# B&R Automation Studio project ConveyorTrackingSolution
Automation Studio 6.3.1.32; technology packages: mappMotion 6.4.1, OpcUaCs 6.3.1

## Configuration Config1

CPU 5APC3100.KBU3-000, AutomationRuntime 6.3.4, Build 11.3.0, Vc 

### Task classes (Cpu.sw)
```
Cyclic#1 (cycle 2000 us, tolerance 0 us):
  MovePrg <- MovePrg.prg
  ParChange <- ParChange.prg
DataObjects: McAcpSys
NcDataObjects: McDriveLog
Binaries: McAcpDrv, udbdef, McAcpSim, TCData, McProfGen, McMechSys, FWRules, ArSvcReg, BRRole, sysconf, iomap, TrkFrmSel, Config_3, Config_9, Config_4, Role, ashwac, Config_10, asfw, Config_5, Config_6, UaCsConfig, Config_8, Config_1, Hierarchy, ashwd, Config_11, Config_7, User, arconfig, Config_2, CommonFeat
Libraries: powerlnk, AsArProf, AsIecCon, fileio, AsIO, UaCoal, AsMem, astime, runtime, AsEPL, DataObj, brsystem, UaCoalPrv, SYS_LIB, MpBase, McBase, MpAxis, McAcpAx, McPathGen, McPureVAx, McAxGroup, McAxis, McProgInt, McTrkPath, MpRobotics
```

### Hardware
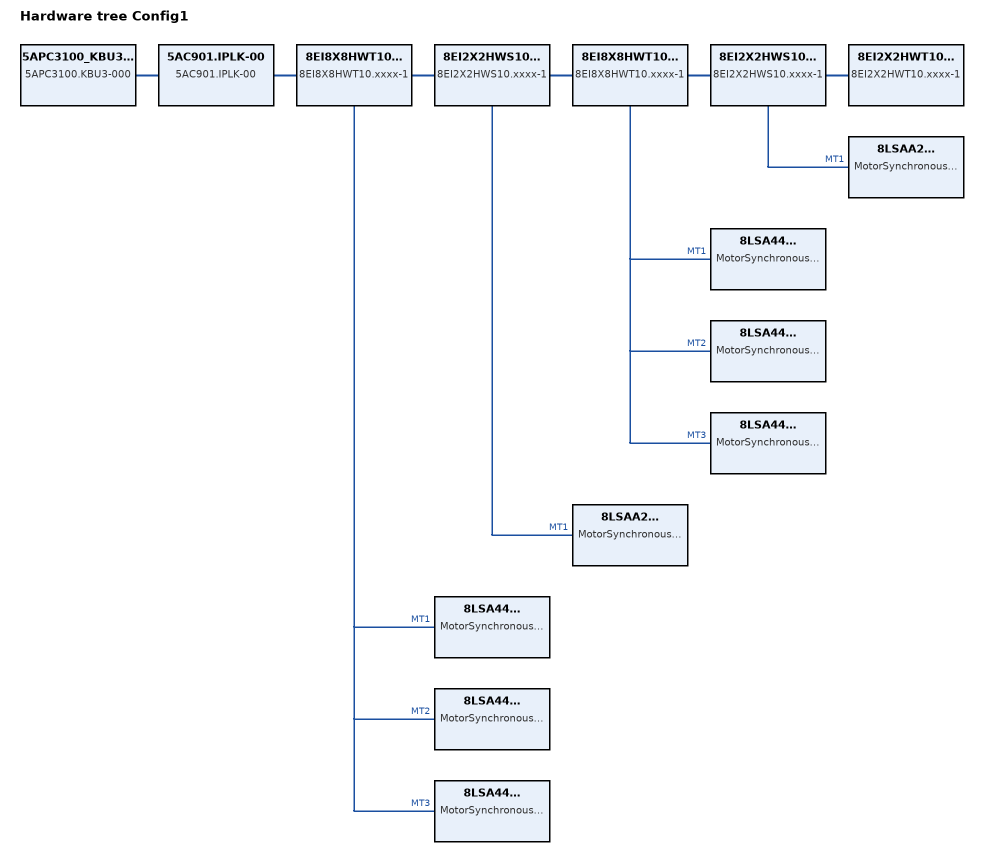
```
5AC901.IPLK-00 : 5AC901.IPLK-00 v2.1.0.0  [SL -> 5APC3100_KBU3_000.SL2]
5APC3100_KBU3_000 : 5APC3100.KBU3-000 v2.2.7.0
  Connector IF3:
    AssignedOperatingSystem = ARemb
    ActivateDevice = 1
  Connector IF4:
    AssignedOperatingSystem = ARemb
    ActivateDevice = 1
  Connector IF5:
    AssignedOperatingSystem = ARemb
  Connector IF6:
    AssignedOperatingSystem = ARemb
  Connector IF7:
    AssignedOperatingSystem = ARemb
  Connector IF8:
    AssignedOperatingSystem = ARemb
  ConfigurationID = ConveyorTrackingSolution_Config1
  Simulation = 1
  Cyclic1Duration = 2000
  Cyclic1Tolerance = 0
  FileDevice1
  FileDeviceName1 = USER
  FileDevicePath1 = USER_PATH
  FileDevice2
  FileDeviceName2 = CNC_PrgDir
  FileDevicePath2 = USER_PATH  // No simulation: use  USER_PATH   ;        Simulation: use    USER_PATH\..\..\..\..\..\Logical\CopyToUserPartition    to directly access the current progam state
8EI2X2HWS10.xxxx-1-QC_D4r1100R_1 : 8EI2X2HWS10.xxxx-1 v2.3.2.0 (NodeNumber=2)  [PLK1 -> 8EI8X8HWT10.xxxx-1-Q1-Q2-Q3_D4r1100R_1.PLK2 [Cable Type=PowerlinkCable, Length=10, Version=1.0.0.3]; PLK2 -> 8EI8X8HWT10.xxxx-1-Q1-Q2-Q3_D4r1100R_2.PLK1 [Cable Type=PowerlinkCable, Length=10, Version=1.0.0.3]]
  DriveConfiguration/Encoder/EncoderX41:
    InterfaceType = EnDat
  DriveConfiguration/Channel[1]/RealAxis:
    AxisReference = gAxisQC_D4r1100R_1
  DriveConfiguration/Channel[1]/RealAxis/MechanicalElements/Gearbox:
    InputIsReadOnly = 1
    Input = 10
    OutputIsReadOnly = 1
  DriveConfiguration/Channel[1]/RealAxis/MechanicalElements/RotaryToLinearTransformation:
    ReferenceDistanceIsReadOnly = 1
    ReferenceDistance = 360
  DriveConfiguration/Channel[1]/RealAxis/Controller:
    ModeIsReadOnly = 1
    Mode = PositionControllerWithTorqueFeedForward
  DriveConfiguration/Channel[1]/RealAxis/Controller/Mode/Position:
    ProportionalGainIsReadOnly = 1
    ProportionalGain = 80.0
    IntegrationTimeIsReadOnly = 1
  DriveConfiguration/Channel[1]/RealAxis/Controller/Mode/Speed:
    ProportionalGainIsReadOnly = 1
    IntegrationTimeIsReadOnly = 1
    FilterTimeIsReadOnly = 1
  DriveConfiguration/Channel[1]/RealAxis/Controller/Mode:
    FeedForwardIsReadOnly = 1
    FeedForward = CyclicValueFromAxesGroup
  DriveConfiguration/Channel[1]/RealAxis/Controller/Mode/LoopFilters:
    LoopFilterXIsReadOnly = 1
  DriveConfiguration/Channel[1]/RealAxis/Homing:
    Mode = Absolute
    RestorePositionVariable = 
  DriveConfiguration/Channel[1]/RealAxis/StopReaction:
    DriveError = CyclicDecelerationFromAxesGroup
  DriveConfiguration/Channel[1]/RealAxis/MovementErrorLimits:
    PositionError = 0.5
  DriveConfiguration/Channel[1]/RealAxis:
    JerkFilterIsReadOnly = 1
    JerkFilter = Used
  DriveConfiguration/Channel[1]/RealAxis/JerkFilter:
    JerkTimeMin = 0.06
    JerkTime = 0.06
8EI2X2HWS10.xxxx-1-QC_D4r1100R_2 : 8EI2X2HWS10.xxxx-1 v2.3.2.0 (NodeNumber=4)  [PLK1 -> 8EI8X8HWT10.xxxx-1-Q1-Q2-Q3_D4r1100R_2.PLK2 [Cable Type=PowerlinkCable, Length=10, Version=1.0.0.3]; PLK2 -> 8EI2X2HWT10.xxxx-1.PLK1 [Cable Type=PowerlinkCable, Length=10, Version=1.0.0.3]]
  DriveConfiguration/Encoder/EncoderX41:
    InterfaceType = EnDat
  DriveConfiguration/Channel[1]/RealAxis:
    AxisReference = gAxisQC_D4r1100R_2
  DriveConfiguration/Channel[1]/RealAxis/MechanicalElements/Gearbox:
    InputIsReadOnly = 1
    Input = 10
    OutputIsReadOnly = 1
  DriveConfiguration/Channel[1]/RealAxis/MechanicalElements/RotaryToLinearTransformation:
    ReferenceDistanceIsReadOnly = 1
    ReferenceDistance = 360
  DriveConfiguration/Channel[1]/RealAxis/Controller:
    ModeIsReadOnly = 1
    Mode = PositionControllerWithTorqueFeedForward
  DriveConfiguration/Channel[1]/RealAxis/Controller/Mode/Position:
    ProportionalGainIsReadOnly = 1
    ProportionalGain = 80.0
    IntegrationTimeIsReadOnly = 1
  DriveConfiguration/Channel[1]/RealAxis/Controller/Mode/Speed:
    ProportionalGainIsReadOnly = 1
    IntegrationTimeIsReadOnly = 1
    FilterTimeIsReadOnly = 1
  DriveConfiguration/Channel[1]/RealAxis/Controller/Mode:
    FeedForwardIsReadOnly = 1
    FeedForward = CyclicValueFromAxesGroup
  DriveConfiguration/Channel[1]/RealAxis/Controller/Mode/LoopFilters:
    LoopFilterXIsReadOnly = 1
  DriveConfiguration/Channel[1]/RealAxis/Homing:
    Mode = Absolute
    RestorePositionVariable = 
  DriveConfiguration/Channel[1]/RealAxis/StopReaction:
    DriveError = CyclicDecelerationFromAxesGroup
  DriveConfiguration/Channel[1]/RealAxis/MovementErrorLimits:
    PositionError = 0.5
  DriveConfiguration/Channel[1]/RealAxis:
    JerkFilterIsReadOnly = 1
    JerkFilter = Used
  DriveConfiguration/Channel[1]/RealAxis/JerkFilter:
    JerkTimeMin = 0.06
    JerkTime = 0.06
8EI2X2HWT10.xxxx-1 : 8EI2X2HWT10.xxxx-1 v2.4.0.0 (NodeNumber=5)  [PLK1 -> 8EI2X2HWS10.xxxx-1-QC_D4r1100R_2.PLK2 [Cable Type=PowerlinkCable, Length=10, Version=1.0.0.3]]
  DriveConfiguration/Channel[1]/RealAxis:
    AxisReference = gAxis_Conveyor_1
  DriveConfiguration/Channel[2]/RealAxis:
    AxisReference = gAxis_Conveyor_2
8EI8X8HWT10.xxxx-1-Q1-Q2-Q3_D4r1100R_1 : 8EI8X8HWT10.xxxx-1 v2.3.2.0 (NodeNumber=1)  [PLK1 -> 5AC901.IPLK-00.IF1 [Cable Type=PowerlinkCable, Length=10, Version=1.0.0.3]; PLK2 -> 8EI2X2HWS10.xxxx-1-QC_D4r1100R_1.PLK1 [Cable Type=PowerlinkCable, Length=10, Version=1.0.0.3]; MT2 -> 8LSA44.DB060S200-3_Q2_D4r1100R_1.MT; MT3 -> 8LSA44.DB060S200-3_Q3_D4r1100R_1.MT]
  DriveConfiguration/Encoder/EncoderX41:
    InterfaceType = EnDat
  DriveConfiguration/Encoder/EncoderX42:
    InterfaceType = EnDat
  DriveConfiguration/Encoder/EncoderX43:
    InterfaceType = EnDat
  DriveConfiguration/Channel[1]/RealAxis:
    AxisReference = gAxisQ1_D4r1100R_1
  DriveConfiguration/Channel[1]/RealAxis/MechanicalElements/Gearbox:
    InputIsReadOnly = 1
    Input = 28
    OutputIsReadOnly = 1
  DriveConfiguration/Channel[1]/RealAxis/MechanicalElements/RotaryToLinearTransformation:
    ReferenceDistanceIsReadOnly = 1
    ReferenceDistance = 360
  DriveConfiguration/Channel[1]/RealAxis/Controller:
    ModeIsReadOnly = 1
    Mode = PositionControllerWithTorqueFeedForward
  DriveConfiguration/Channel[1]/RealAxis/Controller/Mode/Position:
    ProportionalGainIsReadOnly = 1
    ProportionalGain = 150.0
    IntegrationTimeIsReadOnly = 1
  DriveConfiguration/Channel[1]/RealAxis/Controller/Mode/Speed:
    ProportionalGainIsReadOnly = 1
    ProportionalGain = 7.5
    IntegrationTimeIsReadOnly = 1
    FilterTimeIsReadOnly = 1
  DriveConfiguration/Channel[1]/RealAxis/Controller/Mode:
    FeedForwardIsReadOnly = 1
    FeedForward = CyclicValueFromAxesGroup
  DriveConfiguration/Channel[1]/RealAxis/Controller/Mode/LoopFilters:
    LoopFilterXIsReadOnly = 1
  DriveConfiguration/Channel[1]/RealAxis/Homing:
    Mode = Absolute
    RestorePositionVariable = 
  DriveConfiguration/Channel[1]/RealAxis/StopReaction:
    DriveError = CyclicDecelerationFromAxesGroup
  DriveConfiguration/Channel[1]/RealAxis/MovementErrorLimits:
    PositionError = 0.5
  DriveConfiguration/Channel[1]/RealAxis:
    JerkFilterIsReadOnly = 1
    JerkFilter = Used
  DriveConfiguration/Channel[1]/RealAxis/JerkFilter:
    JerkTimeMin = 0.06
    JerkTime = 0.06
  DriveConfiguration/Channel[2]/RealAxis:
    AxisReference = gAxisQ2_D4r1100R_1
  DriveConfiguration/Channel[2]/RealAxis/MechanicalElements/Gearbox:
    InputIsReadOnly = 1
    Input = 28
    OutputIsReadOnly = 1
  DriveConfiguration/Channel[2]/RealAxis/MechanicalElements/RotaryToLinearTransformation:
    ReferenceDistanceIsReadOnly = 1
    ReferenceDistance = 360
  DriveConfiguration/Channel[2]/RealAxis/Controller:
    ModeIsReadOnly = 1
    Mode = PositionControllerWithTorqueFeedForward
  DriveConfiguration/Channel[2]/RealAxis/Controller/Mode/Position:
    ProportionalGainIsReadOnly = 1
    ProportionalGain = 150.0
    IntegrationTimeIsReadOnly = 1
  DriveConfiguration/Channel[2]/RealAxis/Controller/Mode/Speed:
    ProportionalGainIsReadOnly = 1
    ProportionalGain = 7.5
    IntegrationTimeIsReadOnly = 1
    FilterTimeIsReadOnly = 1
  DriveConfiguration/Channel[2]/RealAxis/Controller/Mode:
    FeedForwardIsReadOnly = 1
    FeedForward = CyclicValueFromAxesGroup
  DriveConfiguration/Channel[2]/RealAxis/Controller/Mode/LoopFilters:
    LoopFilterXIsReadOnly = 1
  DriveConfiguration/Channel[2]/RealAxis/Homing:
    Mode = Absolute
    RestorePositionVariable = 
  DriveConfiguration/Channel[2]/RealAxis/StopReaction:
    DriveError = CyclicDecelerationFromAxesGroup
  DriveConfiguration/Channel[2]/RealAxis/MovementErrorLimits:
    PositionError = 0.5
  DriveConfiguration/Channel[2]/RealAxis:
    JerkFilterIsReadOnly = 1
    JerkFilter = Used
  DriveConfiguration/Channel[2]/RealAxis/JerkFilter:
    JerkTimeMin = 0.06
    JerkTime = 0.06
  DriveConfiguration/Channel[3]/RealAxis:
    AxisReference = gAxisQ3_D4r1100R_1
  DriveConfiguration/Channel[3]/RealAxis/MechanicalElements/Gearbox:
    InputIsReadOnly = 1
    Input = 28
    OutputIsReadOnly = 1
  DriveConfiguration/Channel[3]/RealAxis/MechanicalElements/RotaryToLinearTransformation:
    ReferenceDistanceIsReadOnly = 1
    ReferenceDistance = 360
  DriveConfiguration/Channel[3]/RealAxis/Controller:
    ModeIsReadOnly = 1
    Mode = PositionControllerWithTorqueFeedForward
  DriveConfiguration/Channel[3]/RealAxis/Controller/Mode/Position:
    ProportionalGainIsReadOnly = 1
    ProportionalGain = 150.0
    IntegrationTimeIsReadOnly = 1
  DriveConfiguration/Channel[3]/RealAxis/Controller/Mode/Speed:
    ProportionalGainIsReadOnly = 1
    ProportionalGain = 7.5
    IntegrationTimeIsReadOnly = 1
    FilterTimeIsReadOnly = 1
  DriveConfiguration/Channel[3]/RealAxis/Controller/Mode:
    FeedForwardIsReadOnly = 1
    FeedForward = CyclicValueFromAxesGroup
  DriveConfiguration/Channel[3]/RealAxis/Controller/Mode/LoopFilters:
    LoopFilterXIsReadOnly = 1
  DriveConfiguration/Channel[3]/RealAxis/Homing:
    Mode = Absolute
    RestorePositionVariable = 
  DriveConfiguration/Channel[3]/RealAxis/StopReaction:
    DriveError = CyclicDecelerationFromAxesGroup
  DriveConfiguration/Channel[3]/RealAxis/MovementErrorLimits:
    PositionError = 0.5
  DriveConfiguration/Channel[3]/RealAxis:
    JerkFilterIsReadOnly = 1
    JerkFilter = Used
  DriveConfiguration/Channel[3]/RealAxis/JerkFilter:
    JerkTimeMin = 0.06
    JerkTime = 0.06
8EI8X8HWT10.xxxx-1-Q1-Q2-Q3_D4r1100R_2 : 8EI8X8HWT10.xxxx-1 v2.3.2.0 (NodeNumber=3)  [PLK1 -> 8EI2X2HWS10.xxxx-1-QC_D4r1100R_1.PLK2 [Cable Type=PowerlinkCable, Length=10, Version=1.0.0.3]; PLK2 -> 8EI2X2HWS10.xxxx-1-QC_D4r1100R_2.PLK1 [Cable Type=PowerlinkCable, Length=10, Version=1.0.0.3]; MT2 -> 8LSA44.DB060S200-3_Q2_D4r1100R_2.MT; MT3 -> 8LSA44.DB060S200-3_Q3_D4r1100R_2.MT]
  DriveConfiguration/Encoder/EncoderX41:
    InterfaceType = EnDat
  DriveConfiguration/Encoder/EncoderX42:
    InterfaceType = EnDat
  DriveConfiguration/Encoder/EncoderX43:
    InterfaceType = EnDat
  DriveConfiguration/Channel[1]/RealAxis:
    AxisReference = gAxisQ1_D4r1100R_2
  DriveConfiguration/Channel[1]/RealAxis/MechanicalElements/Gearbox:
    InputIsReadOnly = 1
    Input = 28
    OutputIsReadOnly = 1
  DriveConfiguration/Channel[1]/RealAxis/MechanicalElements/RotaryToLinearTransformation:
    ReferenceDistanceIsReadOnly = 1
    ReferenceDistance = 360
  DriveConfiguration/Channel[1]/RealAxis/Controller:
    ModeIsReadOnly = 1
    Mode = PositionControllerWithTorqueFeedForward
  DriveConfiguration/Channel[1]/RealAxis/Controller/Mode/Position:
    ProportionalGainIsReadOnly = 1
    ProportionalGain = 150.0
    IntegrationTimeIsReadOnly = 1
  DriveConfiguration/Channel[1]/RealAxis/Controller/Mode/Speed:
    ProportionalGainIsReadOnly = 1
    ProportionalGain = 7.5
    IntegrationTimeIsReadOnly = 1
    FilterTimeIsReadOnly = 1
  DriveConfiguration/Channel[1]/RealAxis/Controller/Mode:
    FeedForwardIsReadOnly = 1
    FeedForward = CyclicValueFromAxesGroup
  DriveConfiguration/Channel[1]/RealAxis/Controller/Mode/LoopFilters:
    LoopFilterXIsReadOnly = 1
  DriveConfiguration/Channel[1]/RealAxis/Homing:
    Mode = Absolute
    RestorePositionVariable = 
  DriveConfiguration/Channel[1]/RealAxis/StopReaction:
    DriveError = CyclicDecelerationFromAxesGroup
  DriveConfiguration/Channel[1]/RealAxis/MovementErrorLimits:
    PositionError = 0.5
  DriveConfiguration/Channel[1]/RealAxis:
    JerkFilterIsReadOnly = 1
    JerkFilter = Used
  DriveConfiguration/Channel[1]/RealAxis/JerkFilter:
    JerkTimeMin = 0.06
    JerkTime = 0.06
  DriveConfiguration/Channel[2]/RealAxis:
    AxisReference = gAxisQ2_D4r1100R_2
  DriveConfiguration/Channel[2]/RealAxis/MechanicalElements/Gearbox:
    InputIsReadOnly = 1
    Input = 28
    OutputIsReadOnly = 1
  DriveConfiguration/Channel[2]/RealAxis/MechanicalElements/RotaryToLinearTransformation:
    ReferenceDistanceIsReadOnly = 1
    ReferenceDistance = 360
  DriveConfiguration/Channel[2]/RealAxis/Controller:
    ModeIsReadOnly = 1
    Mode = PositionControllerWithTorqueFeedForward
  DriveConfiguration/Channel[2]/RealAxis/Controller/Mode/Position:
    ProportionalGainIsReadOnly = 1
    ProportionalGain = 150.0
    IntegrationTimeIsReadOnly = 1
  DriveConfiguration/Channel[2]/RealAxis/Controller/Mode/Speed:
    ProportionalGainIsReadOnly = 1
    ProportionalGain = 7.5
    IntegrationTimeIsReadOnly = 1
    FilterTimeIsReadOnly = 1
  DriveConfiguration/Channel[2]/RealAxis/Controller/Mode:
    FeedForwardIsReadOnly = 1
    FeedForward = CyclicValueFromAxesGroup
  DriveConfiguration/Channel[2]/RealAxis/Controller/Mode/LoopFilters:
    LoopFilterXIsReadOnly = 1
  DriveConfiguration/Channel[2]/RealAxis/Homing:
    Mode = Absolute
    RestorePositionVariable = 
  DriveConfiguration/Channel[2]/RealAxis/StopReaction:
    DriveError = CyclicDecelerationFromAxesGroup
  DriveConfiguration/Channel[2]/RealAxis/MovementErrorLimits:
    PositionError = 0.5
  DriveConfiguration/Channel[2]/RealAxis:
    JerkFilterIsReadOnly = 1
    JerkFilter = Used
  DriveConfiguration/Channel[2]/RealAxis/JerkFilter:
    JerkTimeMin = 0.06
    JerkTime = 0.06
  DriveConfiguration/Channel[3]/RealAxis:
    AxisReference = gAxisQ3_D4r1100R_2
  DriveConfiguration/Channel[3]/RealAxis/MechanicalElements/Gearbox:
    InputIsReadOnly = 1
    Input = 28
    OutputIsReadOnly = 1
  DriveConfiguration/Channel[3]/RealAxis/MechanicalElements/RotaryToLinearTransformation:
    ReferenceDistanceIsReadOnly = 1
    ReferenceDistance = 360
  DriveConfiguration/Channel[3]/RealAxis/Controller:
    ModeIsReadOnly = 1
    Mode = PositionControllerWithTorqueFeedForward
  DriveConfiguration/Channel[3]/RealAxis/Controller/Mode/Position:
    ProportionalGainIsReadOnly = 1
    ProportionalGain = 150.0
    IntegrationTimeIsReadOnly = 1
  DriveConfiguration/Channel[3]/RealAxis/Controller/Mode/Speed:
    ProportionalGainIsReadOnly = 1
    ProportionalGain = 7.5
    IntegrationTimeIsReadOnly = 1
    FilterTimeIsReadOnly = 1
  DriveConfiguration/Channel[3]/RealAxis/Controller/Mode:
    FeedForwardIsReadOnly = 1
    FeedForward = CyclicValueFromAxesGroup
  DriveConfiguration/Channel[3]/RealAxis/Controller/Mode/LoopFilters:
    LoopFilterXIsReadOnly = 1
  DriveConfiguration/Channel[3]/RealAxis/Homing:
    Mode = Absolute
    RestorePositionVariable = 
  DriveConfiguration/Channel[3]/RealAxis/StopReaction:
    DriveError = CyclicDecelerationFromAxesGroup
  DriveConfiguration/Channel[3]/RealAxis/MovementErrorLimits:
    PositionError = 0.5
  DriveConfiguration/Channel[3]/RealAxis:
    JerkFilterIsReadOnly = 1
    JerkFilter = Used
  DriveConfiguration/Channel[3]/RealAxis/JerkFilter:
    JerkTimeMin = 0.06
    JerkTime = 0.06
8LSA44.DB060S200-3_Q1_D4r1100R_1 : MotorSynchronous_any v2.2.1.0  [MT -> 8EI8X8HWT10.xxxx-1-Q1-Q2-Q3_D4r1100R_1.MT1]
  M1/MotorParameters:
    MOTOR_POLEPAIRS = 5
    MOTOR_SPEED_RATED = 6000
    MOTOR_SPEED_MAX = 12000
    MOTOR_VOLTAGE_RATED = 400
    MOTOR_CURR_RATED = 3.7
    MOTOR_CURR_STALL = 7.4
    MOTOR_CURR_MAX = 43.8
    MOTOR_TORQ_RATED = 3
    MOTOR_TORQ_STALL = 6
    MOTOR_TORQ_MAX = 22.8
    MOTOR_VOLTAGE_CONST = 49.22
    MOTOR_TORQ_CONST = 0.81
    MOTOR_STATOR_RESISTANCE = 0.863
    MOTOR_STATOR_INDUCTANCE = 6.2
    MOTOR_INERTIA = 2.73
    VoltageLimitation = Used
  M1/MotorParameters/VoltageLimitation:
    MOTOR_UDC_MAX = 1000
  M1/MotorParameters/EncoderMounting:
    Angle = StoredOnEncoder
  M1/MotorParameters/TemperatureSensor:
    MOTOR_TEMPSENS_LIM = 130
    TemperatureSensorInterface = EncoderConnectorDigital
    MOTOR_TEMPSENS_PAR1 = 30
    MOTOR_TEMPSENS_PAR2 = 254
    MOTOR_TEMPSENS_PAR3 = -29.72
    MOTOR_TEMPSENS_PAR4 = -4.58
    MOTOR_TEMPSENS_PAR5 = 20.33
    MOTOR_TEMPSENS_PAR6 = 45.18
    MOTOR_TEMPSENS_PAR7 = 69.96
    MOTOR_TEMPSENS_PAR8 = 94.71
    MOTOR_TEMPSENS_PAR9 = 119.6
    MOTOR_TEMPSENS_PAR10 = 149.11
  M1/MotorParameters/TemperatureModel:
    MOTOR_WIND_TEMP_MAX = 110
  M1/MotorParameters/TemperatureModel/Calculation:
    MOTOR_WIND_CROSS_SECT = 0.985
    MOTOR_TAU_THERM = 1800
  M1:
    Brake = Used
  M1/Brake:
    MOTOR_BRAKE_CURR_RATED = 0.83
    MOTOR_BRAKE_TORQ_RATED = 8
    MOTOR_BRAKE_ON_TIME = 0.038
    MOTOR_BRAKE_OFF_TIME = 0.055
    MOTOR_BRAKE_INERTIA = 0.69
  M1/Encoder:
    MOTOR_ENCOD_ATTR = 1
    MOTOR_ENCOD_INERTIA = 0.022
    TemperatureSensor = Used
  M1/Encoder/TemperatureSensor:
    MOTOR_ENCOD_TEMP_LIM = 129
  M1:
    Gearbox = UsedWithDynamicTorqueLimitation
  M1/Gearbox/GearRatio:
    Input = 28
  M1/Gearbox:
    MOTORGEAR_SPEED_MAX = 7500
    MOTORGEAR_TORQ_NOM = 126
    MOTORGEAR_TORQ_MAX = 126
    MOTORGEAR_INERTIA = 0.51
    MOTORGEAR_VISC_FRIC = 0.002
    MOTORGEAR_STAT_FRIC = 0.22
8LSA44.DB060S200-3_Q1_D4r1100R_2 : MotorSynchronous_any v2.2.1.0  [MT -> 8EI8X8HWT10.xxxx-1-Q1-Q2-Q3_D4r1100R_2.MT1]
  M1/MotorParameters:
    MOTOR_POLEPAIRS = 5
    MOTOR_SPEED_RATED = 6000
    MOTOR_SPEED_MAX = 12000
    MOTOR_VOLTAGE_RATED = 400
    MOTOR_CURR_RATED = 3.7
    MOTOR_CURR_STALL = 7.4
    MOTOR_CURR_MAX = 43.8
    MOTOR_TORQ_RATED = 3
    MOTOR_TORQ_STALL = 6
    MOTOR_TORQ_MAX = 22.8
    MOTOR_VOLTAGE_CONST = 49.22
    MOTOR_TORQ_CONST = 0.81
    MOTOR_STATOR_RESISTANCE = 0.863
    MOTOR_STATOR_INDUCTANCE = 6.2
    MOTOR_INERTIA = 2.73
    VoltageLimitation = Used
  M1/MotorParameters/VoltageLimitation:
    MOTOR_UDC_MAX = 1000
  M1/MotorParameters/EncoderMounting:
    Angle = StoredOnEncoder
  M1/MotorParameters/TemperatureSensor:
    MOTOR_TEMPSENS_LIM = 130
    TemperatureSensorInterface = EncoderConnectorDigital
    MOTOR_TEMPSENS_PAR1 = 30
    MOTOR_TEMPSENS_PAR2 = 254
    MOTOR_TEMPSENS_PAR3 = -29.72
    MOTOR_TEMPSENS_PAR4 = -4.58
    MOTOR_TEMPSENS_PAR5 = 20.33
    MOTOR_TEMPSENS_PAR6 = 45.18
    MOTOR_TEMPSENS_PAR7 = 69.96
    MOTOR_TEMPSENS_PAR8 = 94.71
    MOTOR_TEMPSENS_PAR9 = 119.6
    MOTOR_TEMPSENS_PAR10 = 149.11
  M1/MotorParameters/TemperatureModel:
    MOTOR_WIND_TEMP_MAX = 110
  M1/MotorParameters/TemperatureModel/Calculation:
    MOTOR_WIND_CROSS_SECT = 0.985
    MOTOR_TAU_THERM = 1800
  M1:
    Brake = Used
  M1/Brake:
    MOTOR_BRAKE_CURR_RATED = 0.83
    MOTOR_BRAKE_TORQ_RATED = 8
    MOTOR_BRAKE_ON_TIME = 0.038
    MOTOR_BRAKE_OFF_TIME = 0.055
    MOTOR_BRAKE_INERTIA = 0.69
  M1/Encoder:
    MOTOR_ENCOD_ATTR = 1
    MOTOR_ENCOD_INERTIA = 0.022
    TemperatureSensor = Used
  M1/Encoder/TemperatureSensor:
    MOTOR_ENCOD_TEMP_LIM = 129
  M1:
    Gearbox = UsedWithDynamicTorqueLimitation
  M1/Gearbox/GearRatio:
    Input = 28
  M1/Gearbox:
    MOTORGEAR_SPEED_MAX = 7500
    MOTORGEAR_TORQ_NOM = 126
    MOTORGEAR_TORQ_MAX = 126
    MOTORGEAR_INERTIA = 0.51
    MOTORGEAR_VISC_FRIC = 0.002
    MOTORGEAR_STAT_FRIC = 0.22
8LSA44.DB060S200-3_Q2_D4r1100R_1 : MotorSynchronous_any v2.2.1.0  [MT -> 8EI8X8HWT10.xxxx-1-Q1-Q2-Q3_D4r1100R_1.MT2]
  M1/MotorParameters:
    MOTOR_POLEPAIRS = 5
    MOTOR_SPEED_RATED = 6000
    MOTOR_SPEED_MAX = 12000
    MOTOR_VOLTAGE_RATED = 400
    MOTOR_CURR_RATED = 3.7
    MOTOR_CURR_STALL = 7.4
    MOTOR_CURR_MAX = 43.8
    MOTOR_TORQ_RATED = 3
    MOTOR_TORQ_STALL = 6
    MOTOR_TORQ_MAX = 22.8
    MOTOR_VOLTAGE_CONST = 49.22
    MOTOR_TORQ_CONST = 0.81
    MOTOR_STATOR_RESISTANCE = 0.863
    MOTOR_STATOR_INDUCTANCE = 6.2
    MOTOR_INERTIA = 2.73
    VoltageLimitation = Used
  M1/MotorParameters/VoltageLimitation:
    MOTOR_UDC_MAX = 1000
  M1/MotorParameters/EncoderMounting:
    Angle = StoredOnEncoder
  M1/MotorParameters/TemperatureSensor:
    MOTOR_TEMPSENS_LIM = 130
    TemperatureSensorInterface = EncoderConnectorDigital
    MOTOR_TEMPSENS_PAR1 = 30
    MOTOR_TEMPSENS_PAR2 = 254
    MOTOR_TEMPSENS_PAR3 = -29.72
    MOTOR_TEMPSENS_PAR4 = -4.58
    MOTOR_TEMPSENS_PAR5 = 20.33
    MOTOR_TEMPSENS_PAR6 = 45.18
    MOTOR_TEMPSENS_PAR7 = 69.96
    MOTOR_TEMPSENS_PAR8 = 94.71
    MOTOR_TEMPSENS_PAR9 = 119.6
    MOTOR_TEMPSENS_PAR10 = 149.11
  M1/MotorParameters/TemperatureModel:
    MOTOR_WIND_TEMP_MAX = 110
  M1/MotorParameters/TemperatureModel/Calculation:
    MOTOR_WIND_CROSS_SECT = 0.985
    MOTOR_TAU_THERM = 1800
  M1:
    Brake = Used
  M1/Brake:
    MOTOR_BRAKE_CURR_RATED = 0.83
    MOTOR_BRAKE_TORQ_RATED = 8
    MOTOR_BRAKE_ON_TIME = 0.038
    MOTOR_BRAKE_OFF_TIME = 0.055
    MOTOR_BRAKE_INERTIA = 0.69
  M1/Encoder:
    MOTOR_ENCOD_ATTR = 1
    MOTOR_ENCOD_INERTIA = 0.022
    TemperatureSensor = Used
  M1/Encoder/TemperatureSensor:
    MOTOR_ENCOD_TEMP_LIM = 129
  M1:
    Gearbox = UsedWithDynamicTorqueLimitation
  M1/Gearbox/GearRatio:
    Input = 28
  M1/Gearbox:
    MOTORGEAR_SPEED_MAX = 7500
    MOTORGEAR_TORQ_NOM = 126
    MOTORGEAR_TORQ_MAX = 126
    MOTORGEAR_INERTIA = 0.51
    MOTORGEAR_VISC_FRIC = 0.002
    MOTORGEAR_STAT_FRIC = 0.22
8LSA44.DB060S200-3_Q2_D4r1100R_2 : MotorSynchronous_any v2.2.1.0  [MT -> 8EI8X8HWT10.xxxx-1-Q1-Q2-Q3_D4r1100R_2.MT2]
  M1/MotorParameters:
    MOTOR_POLEPAIRS = 5
    MOTOR_SPEED_RATED = 6000
    MOTOR_SPEED_MAX = 12000
    MOTOR_VOLTAGE_RATED = 400
    MOTOR_CURR_RATED = 3.7
    MOTOR_CURR_STALL = 7.4
    MOTOR_CURR_MAX = 43.8
    MOTOR_TORQ_RATED = 3
    MOTOR_TORQ_STALL = 6
    MOTOR_TORQ_MAX = 22.8
    MOTOR_VOLTAGE_CONST = 49.22
    MOTOR_TORQ_CONST = 0.81
    MOTOR_STATOR_RESISTANCE = 0.863
    MOTOR_STATOR_INDUCTANCE = 6.2
    MOTOR_INERTIA = 2.73
    VoltageLimitation = Used
  M1/MotorParameters/VoltageLimitation:
    MOTOR_UDC_MAX = 1000
  M1/MotorParameters/EncoderMounting:
    Angle = StoredOnEncoder
  M1/MotorParameters/TemperatureSensor:
    MOTOR_TEMPSENS_LIM = 130
    TemperatureSensorInterface = EncoderConnectorDigital
    MOTOR_TEMPSENS_PAR1 = 30
    MOTOR_TEMPSENS_PAR2 = 254
    MOTOR_TEMPSENS_PAR3 = -29.72
    MOTOR_TEMPSENS_PAR4 = -4.58
    MOTOR_TEMPSENS_PAR5 = 20.33
    MOTOR_TEMPSENS_PAR6 = 45.18
    MOTOR_TEMPSENS_PAR7 = 69.96
    MOTOR_TEMPSENS_PAR8 = 94.71
    MOTOR_TEMPSENS_PAR9 = 119.6
    MOTOR_TEMPSENS_PAR10 = 149.11
  M1/MotorParameters/TemperatureModel:
    MOTOR_WIND_TEMP_MAX = 110
  M1/MotorParameters/TemperatureModel/Calculation:
    MOTOR_WIND_CROSS_SECT = 0.985
    MOTOR_TAU_THERM = 1800
  M1:
    Brake = Used
  M1/Brake:
    MOTOR_BRAKE_CURR_RATED = 0.83
    MOTOR_BRAKE_TORQ_RATED = 8
    MOTOR_BRAKE_ON_TIME = 0.038
    MOTOR_BRAKE_OFF_TIME = 0.055
    MOTOR_BRAKE_INERTIA = 0.69
  M1/Encoder:
    MOTOR_ENCOD_ATTR = 1
    MOTOR_ENCOD_INERTIA = 0.022
    TemperatureSensor = Used
  M1/Encoder/TemperatureSensor:
    MOTOR_ENCOD_TEMP_LIM = 129
  M1:
    Gearbox = UsedWithDynamicTorqueLimitation
  M1/Gearbox/GearRatio:
    Input = 28
  M1/Gearbox:
    MOTORGEAR_SPEED_MAX = 7500
    MOTORGEAR_TORQ_NOM = 126
    MOTORGEAR_TORQ_MAX = 126
    MOTORGEAR_INERTIA = 0.51
    MOTORGEAR_VISC_FRIC = 0.002
    MOTORGEAR_STAT_FRIC = 0.22
8LSA44.DB060S200-3_Q3_D4r1100R_1 : MotorSynchronous_any v2.2.1.0  [MT -> 8EI8X8HWT10.xxxx-1-Q1-Q2-Q3_D4r1100R_1.MT3]
  M1/MotorParameters:
    MOTOR_POLEPAIRS = 5
    MOTOR_SPEED_RATED = 6000
    MOTOR_SPEED_MAX = 12000
    MOTOR_VOLTAGE_RATED = 400
    MOTOR_CURR_RATED = 3.7
    MOTOR_CURR_STALL = 7.4
    MOTOR_CURR_MAX = 43.8
    MOTOR_TORQ_RATED = 3
    MOTOR_TORQ_STALL = 6
    MOTOR_TORQ_MAX = 22.8
    MOTOR_VOLTAGE_CONST = 49.22
    MOTOR_TORQ_CONST = 0.81
    MOTOR_STATOR_RESISTANCE = 0.863
    MOTOR_STATOR_INDUCTANCE = 6.2
    MOTOR_INERTIA = 2.73
    VoltageLimitation = Used
  M1/MotorParameters/VoltageLimitation:
    MOTOR_UDC_MAX = 1000
  M1/MotorParameters/EncoderMounting:
    Angle = StoredOnEncoder
  M1/MotorParameters/TemperatureSensor:
    MOTOR_TEMPSENS_LIM = 130
    TemperatureSensorInterface = EncoderConnectorDigital
    MOTOR_TEMPSENS_PAR1 = 30
    MOTOR_TEMPSENS_PAR2 = 254
    MOTOR_TEMPSENS_PAR3 = -29.72
    MOTOR_TEMPSENS_PAR4 = -4.58
    MOTOR_TEMPSENS_PAR5 = 20.33
    MOTOR_TEMPSENS_PAR6 = 45.18
    MOTOR_TEMPSENS_PAR7 = 69.96
    MOTOR_TEMPSENS_PAR8 = 94.71
    MOTOR_TEMPSENS_PAR9 = 119.6
    MOTOR_TEMPSENS_PAR10 = 149.11
  M1/MotorParameters/TemperatureModel:
    MOTOR_WIND_TEMP_MAX = 110
  M1/MotorParameters/TemperatureModel/Calculation:
    MOTOR_WIND_CROSS_SECT = 0.985
    MOTOR_TAU_THERM = 1800
  M1:
    Brake = Used
  M1/Brake:
    MOTOR_BRAKE_CURR_RATED = 0.83
    MOTOR_BRAKE_TORQ_RATED = 8
    MOTOR_BRAKE_ON_TIME = 0.038
    MOTOR_BRAKE_OFF_TIME = 0.055
    MOTOR_BRAKE_INERTIA = 0.69
  M1/Encoder:
    MOTOR_ENCOD_ATTR = 1
    MOTOR_ENCOD_INERTIA = 0.022
    TemperatureSensor = Used
  M1/Encoder/TemperatureSensor:
    MOTOR_ENCOD_TEMP_LIM = 129
  M1:
    Gearbox = UsedWithDynamicTorqueLimitation
  M1/Gearbox/GearRatio:
    Input = 28
  M1/Gearbox:
    MOTORGEAR_SPEED_MAX = 7500
    MOTORGEAR_TORQ_NOM = 126
    MOTORGEAR_TORQ_MAX = 126
    MOTORGEAR_INERTIA = 0.51
    MOTORGEAR_VISC_FRIC = 0.002
    MOTORGEAR_STAT_FRIC = 0.22
8LSA44.DB060S200-3_Q3_D4r1100R_2 : MotorSynchronous_any v2.2.1.0  [MT -> 8EI8X8HWT10.xxxx-1-Q1-Q2-Q3_D4r1100R_2.MT3]
  M1/MotorParameters:
    MOTOR_POLEPAIRS = 5
    MOTOR_SPEED_RATED = 6000
    MOTOR_SPEED_MAX = 12000
    MOTOR_VOLTAGE_RATED = 400
    MOTOR_CURR_RATED = 3.7
    MOTOR_CURR_STALL = 7.4
    MOTOR_CURR_MAX = 43.8
    MOTOR_TORQ_RATED = 3
    MOTOR_TORQ_STALL = 6
    MOTOR_TORQ_MAX = 22.8
    MOTOR_VOLTAGE_CONST = 49.22
    MOTOR_TORQ_CONST = 0.81
    MOTOR_STATOR_RESISTANCE = 0.863
    MOTOR_STATOR_INDUCTANCE = 6.2
    MOTOR_INERTIA = 2.73
    VoltageLimitation = Used
  M1/MotorParameters/VoltageLimitation:
    MOTOR_UDC_MAX = 1000
  M1/MotorParameters/EncoderMounting:
    Angle = StoredOnEncoder
  M1/MotorParameters/TemperatureSensor:
    MOTOR_TEMPSENS_LIM = 130
    TemperatureSensorInterface = EncoderConnectorDigital
    MOTOR_TEMPSENS_PAR1 = 30
    MOTOR_TEMPSENS_PAR2 = 254
    MOTOR_TEMPSENS_PAR3 = -29.72
    MOTOR_TEMPSENS_PAR4 = -4.58
    MOTOR_TEMPSENS_PAR5 = 20.33
    MOTOR_TEMPSENS_PAR6 = 45.18
    MOTOR_TEMPSENS_PAR7 = 69.96
    MOTOR_TEMPSENS_PAR8 = 94.71
    MOTOR_TEMPSENS_PAR9 = 119.6
    MOTOR_TEMPSENS_PAR10 = 149.11
  M1/MotorParameters/TemperatureModel:
    MOTOR_WIND_TEMP_MAX = 110
  M1/MotorParameters/TemperatureModel/Calculation:
    MOTOR_WIND_CROSS_SECT = 0.985
    MOTOR_TAU_THERM = 1800
  M1:
    Brake = Used
  M1/Brake:
    MOTOR_BRAKE_CURR_RATED = 0.83
    MOTOR_BRAKE_TORQ_RATED = 8
    MOTOR_BRAKE_ON_TIME = 0.038
    MOTOR_BRAKE_OFF_TIME = 0.055
    MOTOR_BRAKE_INERTIA = 0.69
  M1/Encoder:
    MOTOR_ENCOD_ATTR = 1
    MOTOR_ENCOD_INERTIA = 0.022
    TemperatureSensor = Used
  M1/Encoder/TemperatureSensor:
    MOTOR_ENCOD_TEMP_LIM = 129
  M1:
    Gearbox = UsedWithDynamicTorqueLimitation
  M1/Gearbox/GearRatio:
    Input = 28
  M1/Gearbox:
    MOTORGEAR_SPEED_MAX = 7500
    MOTORGEAR_TORQ_NOM = 126
    MOTORGEAR_TORQ_MAX = 126
    MOTORGEAR_INERTIA = 0.51
    MOTORGEAR_VISC_FRIC = 0.002
    MOTORGEAR_STAT_FRIC = 0.22
8LSAA2.D9045S200-3_QC_D4r1100R_1 : MotorSynchronous_any v2.2.1.0  [MT -> 8EI2X2HWS10.xxxx-1-QC_D4r1100R_1.MT1]
  M1/MotorParameters:
    MOTOR_POLEPAIRS = 5
    MOTOR_SPEED_RATED = 4500
    MOTOR_SPEED_MAX = 7000
    MOTOR_VOLTAGE_RATED = 400
    MOTOR_CURR_RATED = 1.31
    MOTOR_CURR_STALL = 1.42
    MOTOR_CURR_MAX = 6
    MOTOR_TORQ_RATED = 1.27
    MOTOR_TORQ_STALL = 1.4
    MOTOR_TORQ_MAX = 4.5
    MOTOR_VOLTAGE_CONST = 58.64
    MOTOR_TORQ_CONST = 0.97
    MOTOR_STATOR_RESISTANCE = 13.9
    MOTOR_STATOR_INDUCTANCE = 27
    MOTOR_INERTIA = 0.38
    VoltageLimitation = Used
  M1/MotorParameters/VoltageLimitation:
    MOTOR_UDC_MAX = 1000
  M1/MotorParameters/EncoderMounting:
    Angle = StoredOnEncoder
  M1/MotorParameters/TemperatureSensor:
    MOTOR_TEMPSENS_LIM = 130
    TemperatureSensorInterface = EncoderConnectorDigital
    MOTOR_TEMPSENS_PAR1 = 30
    MOTOR_TEMPSENS_PAR2 = 254
    MOTOR_TEMPSENS_PAR3 = -29.72
    MOTOR_TEMPSENS_PAR4 = -4.58
    MOTOR_TEMPSENS_PAR5 = 20.33
    MOTOR_TEMPSENS_PAR6 = 45.18
    MOTOR_TEMPSENS_PAR7 = 69.96
    MOTOR_TEMPSENS_PAR8 = 94.71
    MOTOR_TEMPSENS_PAR9 = 119.6
    MOTOR_TEMPSENS_PAR10 = 149.11
  M1/MotorParameters/TemperatureModel:
    MOTOR_WIND_TEMP_MAX = 110
  M1/MotorParameters/TemperatureModel/Calculation:
    MOTOR_WIND_CROSS_SECT = 0.126
    MOTOR_TAU_THERM = 1860
  M1:
    Brake = Used
  M1/Brake:
    MOTOR_BRAKE_CURR_RATED = 0.56
    MOTOR_BRAKE_TORQ_RATED = 3.2
    MOTOR_BRAKE_ON_TIME = 0.01
    MOTOR_BRAKE_OFF_TIME = 0.06
    MOTOR_BRAKE_INERTIA = 0.38
  M1/Encoder:
    MOTOR_ENCOD_ATTR = 1
    MOTOR_ENCOD_INERTIA = 0.004
    TemperatureSensor = Used
  M1/Encoder/TemperatureSensor:
    MOTOR_ENCOD_TEMP_LIM = 124
  M1:
    Gearbox = UsedWithDynamicTorqueLimitation
  M1/Gearbox/GearRatio:
    Input = 10
  M1/Gearbox:
    MOTORGEAR_SPEED_MAX = 7500
    MOTORGEAR_TORQ_NOM = 7.0
    MOTORGEAR_TORQ_MAX = 7.0
    MOTORGEAR_INERTIA = 0.16
    MOTORGEAR_VISC_FRIC = 0.0038
    MOTORGEAR_STAT_FRIC = 0.07
8LSAA2.D9045S200-3_QC_D4r1100R_2 : MotorSynchronous_any v2.2.1.0  [MT -> 8EI2X2HWS10.xxxx-1-QC_D4r1100R_2.MT1]
  M1/MotorParameters:
    MOTOR_POLEPAIRS = 5
    MOTOR_SPEED_RATED = 4500
    MOTOR_SPEED_MAX = 7000
    MOTOR_VOLTAGE_RATED = 400
    MOTOR_CURR_RATED = 1.31
    MOTOR_CURR_STALL = 1.42
    MOTOR_CURR_MAX = 6
    MOTOR_TORQ_RATED = 1.27
    MOTOR_TORQ_STALL = 1.4
    MOTOR_TORQ_MAX = 4.5
    MOTOR_VOLTAGE_CONST = 58.64
    MOTOR_TORQ_CONST = 0.97
    MOTOR_STATOR_RESISTANCE = 13.9
    MOTOR_STATOR_INDUCTANCE = 27
    MOTOR_INERTIA = 0.38
    VoltageLimitation = Used
  M1/MotorParameters/VoltageLimitation:
    MOTOR_UDC_MAX = 1000
  M1/MotorParameters/EncoderMounting:
    Angle = StoredOnEncoder
  M1/MotorParameters/TemperatureSensor:
    MOTOR_TEMPSENS_LIM = 130
    TemperatureSensorInterface = EncoderConnectorDigital
    MOTOR_TEMPSENS_PAR1 = 30
    MOTOR_TEMPSENS_PAR2 = 254
    MOTOR_TEMPSENS_PAR3 = -29.72
    MOTOR_TEMPSENS_PAR4 = -4.58
    MOTOR_TEMPSENS_PAR5 = 20.33
    MOTOR_TEMPSENS_PAR6 = 45.18
    MOTOR_TEMPSENS_PAR7 = 69.96
    MOTOR_TEMPSENS_PAR8 = 94.71
    MOTOR_TEMPSENS_PAR9 = 119.6
    MOTOR_TEMPSENS_PAR10 = 149.11
  M1/MotorParameters/TemperatureModel:
    MOTOR_WIND_TEMP_MAX = 110
  M1/MotorParameters/TemperatureModel/Calculation:
    MOTOR_WIND_CROSS_SECT = 0.126
    MOTOR_TAU_THERM = 1860
  M1:
    Brake = Used
  M1/Brake:
    MOTOR_BRAKE_CURR_RATED = 0.56
    MOTOR_BRAKE_TORQ_RATED = 3.2
    MOTOR_BRAKE_ON_TIME = 0.01
    MOTOR_BRAKE_OFF_TIME = 0.06
    MOTOR_BRAKE_INERTIA = 0.38
  M1/Encoder:
    MOTOR_ENCOD_ATTR = 1
    MOTOR_ENCOD_INERTIA = 0.004
    TemperatureSensor = Used
  M1/Encoder/TemperatureSensor:
    MOTOR_ENCOD_TEMP_LIM = 124
  M1:
    Gearbox = UsedWithDynamicTorqueLimitation
  M1/Gearbox/GearRatio:
    Input = 10
  M1/Gearbox:
    MOTORGEAR_SPEED_MAX = 7500
    MOTORGEAR_TORQ_NOM = 7.0
    MOTORGEAR_TORQ_MAX = 7.0
    MOTORGEAR_INERTIA = 0.16
    MOTORGEAR_VISC_FRIC = 0.0038
    MOTORGEAR_STAT_FRIC = 0.07
```

### Config_5.axis - 5APC3100_KBU3_000/mappMotion/ConveyorBelts/Config_5.axis
```
Element gAxis_Conveyor_1 (Type=axis)
  BaseType = LinearPeriodic
    PeriodSettings:
      Period = 4000
  MovementLimits:
    Acceleration:
      Acceleration = 500
    Deceleration:
      Deceleration = 500
Element gAxis_Conveyor_2 (Type=axis)
  BaseType = LinearPeriodic
    PeriodSettings:
      Period = 4000
  MovementLimits:
    Acceleration:
      Acceleration = 500
    Deceleration:
      Deceleration = 500
```

### Config_6.trackingpath - 5APC3100_KBU3_000/mappMotion/ConveyorBelts/Config_6.trackingpath
```
Element gTrkPath_Conveyor_1 (Type=trackingpath)
  Type:
    MaxTrackingFrames = 10000
    MotionSource = Axis
      AxisRef = gAxis_Conveyor_1
    TrackingFrames:
      AutomaticCreation:
        Condition[1]:
          Distance = 150
      AutomaticDeletion:
        Condition[1]:
          MinPosition = 0
          MaxPosition = 3000
        Condition[2] = AfterDesynchronization
          AxesGroupRef = gAxesGroup_D4r1100R_1
        Condition[3] = AfterDesynchronization
          AxesGroupRef = gAxesGroup_D4r1100R_2
  SceneViewerObject:
    VisualRepresentation = Conveyor belt
      Dimensions:
        Length = 3000
        Width = 200
        Height = 50
      Translation:
        Y = -100
        Z = -50
      Material = GreyMatte
Element gTrkPath_Conveyor_2 (Type=trackingpath)
  Type:
    MaxTrackingFrames = 10000
    MotionSource = Axis
      AxisRef = gAxis_Conveyor_2
    TrackingFrames:
      AutomaticCreation:
        Condition[1]:
          Distance = 150
      AutomaticDeletion:
        Condition[1]:
          MinPosition = 0
          MaxPosition = 3000
        Condition[2] = AfterDesynchronization
          AxesGroupRef = gAxesGroup_D4r1100R_1
        Condition[3] = AfterDesynchronization
          AxesGroupRef = gAxesGroup_D4r1100R_2
  SceneViewerObject:
    VisualRepresentation = Conveyor belt
      Dimensions:
        Length = 3000
        Width = 200
        Height = 50
      Translation:
        Y = -100
        Z = -50
      Material = GreyMatte
```

### Config_1.axesgroup - 5APC3100_KBU3_000/mappMotion/Robots/Codian_D4r1100R_1/Config_1.axesgroup
```
Element gAxesGroup_D4r1100R_1 (Type=axesgroup)
  Type = PathGenAxesGroup
    ProcessingTaskClass = 1
    PhysicalAxes:
      JointAxes:
        JointAxis[1]:
          AxisRef = gAxisQ1_D4r1100R_1
        JointAxis[2]:
          AxisRef = gAxisQ2_D4r1100R_1
        JointAxis[3]:
          AxisRef = gAxisQ3_D4r1100R_1
        JointAxis[4]:
          Name = QC
          AxisRef = gAxisQC_D4r1100R_1
    MechanicalSystem:
      MechSysRef = MechSys_D4r1100R_1
    BasicSettings:
      GeometryPlanning:
        MaxTangentialTransitionDeviation = 0.05
      TrajectoryPlanning:
        LimitCheckResolution:
          Time = 0.005
        BufferTime:
          Time = 0.05
      Miscellaneous:
        TimeStretchOverride:
          JerkSuppression = Basic
            AdaptationTime = 0.3
    StopReaction:
      AxisError:
        AxisReaction = DynamicStop
    AxesGroupFeatures:
      FeatureRef[1] = Feature_Programs_D4r1100R_1
      FeatureRef[2] = Feature_FeedForward_D4r1100R_X
      FeatureRef[3] = Feature_Jogging_D4r1100R_X
      FeatureRef[4] = Feature_PathDefinitions_D4r1100R_X
      FeatureRef[5] = Feature_TrkFrmSel_D4r1100R_X
      FeatureRef[6] = Feature_Tracking_D4r1100R_X
```

### Config_4.axesgroupfeature - 5APC3100_KBU3_000/mappMotion/Robots/Codian_D4r1100R_1/Config_4.axesgroupfeature
```
Element Feature_Programs_D4r1100R_1 (Type=axesgroupfeature)
  Type:
    ProgramElements:
      PVs:
        PV[1]:
          PvName = ::MovePrg:GripperRobot1OpenClose
          Advanced:
            Alias = CloseGripper
            Synchronization = Path
```

### Config_10.mechanicalsystem - 5APC3100_KBU3_000/mappMotion/Robots/Codian_D4r1100R_2/Config_10.mechanicalsystem
```
Element MechSys_D4r1100R_2 (Type=mechanicalsystem)
  TypeIsReadOnly = 1
  Type = Delta
    SubtypeIsReadOnly = 1
    Subtype = 4AxesDeltaA
      SceneViewerObject = ObjectID
        ID = 1790
      DescriptionIsReadOnly = 1
      Description:
        Dimensions:
          BasePlatform:
            ArmLinkPointIsReadOnly = 1
            Arm1LinkPoint:
              Radius = 200.0
              Z = -90.0
            Arm2LinkPoint:
              Angle = -120.0
              Radius = 200.0
              Z = -90.0
            Arm3LinkPoint:
              Angle = -240.0
              Radius = 200.0
              Z = -90.0
          Arms:
            ArmIsReadOnly = 1
            Arm1:
              UpperArmLength = 320.0
              LowerArmLength = 850.0
            Arm2:
              UpperArmLength = 320.0
              LowerArmLength = 850.0
            Arm3:
              UpperArmLength = 320.0
              LowerArmLength = 850.0
            LowerArmPairDistance = 104.0
          EndEffectorPlatform:
            ArmLinkPointIsReadOnly = 1
            Arm1LinkPoint:
              Radius = 50.0
            Arm2LinkPoint:
              Radius = 50.0
            Arm3LinkPoint:
              Radius = 50.0
            TranslationToFlange:
              Z = -32.6
        Offsets:
          JointAxisIsReadOnly = 1
          JointAxis[1]
          JointAxis[2]
          JointAxis[3]
          JointAxis[4]
        CountDirections:
          JointAxisIsReadOnly = 1
          JointAxis[1]
          JointAxis[2]
          JointAxis[3]
          JointAxis[4]
      TcpOrientation:
        Frames = Used
      WireFrameModel:
        UpperArm1:
          Distance = 5
        LowerArm1:
          Distance = 5
        UpperArm2:
          Distance = 5
        LowerArm2:
          Distance = 5
        UpperArm3:
          Distance = 5
        LowerArm3:
          Distance = 5
        EndEffectorPlatformToFlange:
          Distance = 5
        FlangeToTcp = NotUsed
      DynamicModelIsReadOnly = 1
      InternalDynamicModelIsReadOnly = 1
      InternalDynamicModel = Used
        TypeIsReadOnly = 1
        Type = D4-ST21-1100-R11
        Row[1]:
          Value = 4
          Unit = Variant
          Description = Type of dynamic model
        Row[2]:
          Index = 1
          Value = 1.017
          Unit = 
          Description = m1
        Row[3]:
          Index = 2
          Value = 0.10420181999999999
          Unit = 
          Description = m1*rc1x
        Row[4]:
          Index = 3
          Unit = 
          Description = m1*rc1y
        Row[5]:
          Index = 4
          Value = 0.00444429
          Unit = 
          Description = m1*rc1z
        Row[6]:
          Index = 5
          Unit = 
          Description = m1*rc1x*rc1y
        Row[7]:
          Index = 6
          Unit = 
          Description = m1*rc1y*rc1z
        Row[8]:
          Index = 7
          Value = 0.0004553619534
          Unit = 
          Description = m1*rc1x*rc1z
        Row[9]:
          Index = 8
          Value = 0.010676518477199998
          Unit = 
          Description = m1*rc1x^2
        Row[10]:
          Index = 9
          Unit = 
          Description = m1*rc1y^2
        Row[11]:
          Index = 10
          Value = 1.9421547300000004e-05
          Unit = 
          Description = m1*rc1z^2
        Row[12]:
          Index = 11
          Unit = 
          Description = Jxx1
        Row[13]:
          Index = 12
          Value = 0.012935562
          Unit = 
          Description = Jyy1
        Row[14]:
          Index = 13
          Unit = 
          Description = Jzz1
        Row[15]:
          Index = 14
          Value = 1.017
          Unit = 
          Description = m2
        Row[16]:
          Index = 15
          Value = 0.10420181999999999
          Unit = 
          Description = m2*rc2x
        Row[17]:
          Index = 16
          Unit = 
          Description = m2*rc2y
        Row[18]:
          Index = 17
          Value = 0.00444429
          Unit = 
          Description = m2*rc2z
        Row[19]:
          Index = 18
          Unit = 
          Description = m2*rc2x*rc2y
        Row[20]:
          Index = 19
          Unit = 
          Description = m2*rc2y*rc2z
        Row[21]:
          Index = 20
          Value = 0.0004553619534
          Unit = 
          Description = m2*rc2x*rc2z
        Row[22]:
          Index = 21
          Value = 0.010676518477199998
          Unit = 
          Description = m2*rc2x^2
        Row[23]:
          Index = 22
          Unit = 
          Description = m2*rc2y^2
        Row[24]:
          Index = 23
          Value = 1.9421547300000004e-05
          Unit = 
          Description = m2*rc2z^2
        Row[25]:
          Index = 24
          Unit = 
          Description = Jxx2
        Row[26]:
          Index = 25
          Value = 0.012935562
          Unit = 
          Description = Jyy2
        Row[27]:
          Index = 26
          Unit = 
          Description = Jzz2
        Row[28]:
          Index = 27
          Value = 1.017
          Unit = 
          Description = m3
        Row[29]:
          Index = 28
          Value = 0.10420181999999999
          Unit = 
          Description = m3*rc3x
        Row[30]:
          Index = 29
          Unit = 
          Description = m3*rc3y
        Row[31]:
          Index = 30
          Value = 0.00444429
          Unit = 
          Description = m3*rc3z
        Row[32]:
          Index = 31
          Unit = 
          Description = m3*rc3x*rc3y
        Row[33]:
          Index = 32
          Unit = 
          Description = m3*rc3y*rc3z
        Row[34]:
          Index = 33
          Value = 0.0004553619534
          Unit = 
          Description = m3*rc3x*rc3z
        Row[35]:
          Index = 34
          Value = 0.010676518477199998
          Unit = 
          Description = m3*rc3x^2
        Row[36]:
          Index = 35
          Unit = 
          Description = m3*rc3y^2
        Row[37]:
          Index = 36
          Value = 1.9421547300000004e-05
          Unit = 
          Description = m3*rc3z^2
        Row[38]:
          Index = 37
          Unit = 
          Description = Jxx3
        Row[39]:
          Index = 38
          Value = 0.012935562
          Unit = 
          Description = Jyy3
        Row[40]:
          Index = 39
          Unit = 
          Description = Jzz3
        Row[41]:
          Index = 40
          Value = 0.363
          Unit = 
          Description = m4
        Row[42]:
          Index = 41
          Unit = 
          Description = m4*rc4x
        Row[43]:
          Index = 42
          Unit = 
          Description = m4*rc4y
        Row[44]:
          Index = 43
          Value = 0.154275
          Unit = 
          Description = m4*rc4z
        Row[45]:
          Index = 44
          Unit = 
          Description = m4*rc4x*rc4y
        Row[46]:
          Index = 45
          Unit = 
          Description = m4*rc4y*rc4z
        Row[47]:
          Index = 46
          Unit = 
          Description = m4*rc4x*rc4z
        Row[48]:
          Index = 47
          Unit = 
          Description = m4*rc4x^2
        Row[49]:
          Index = 48
          Unit = 
          Description = m4*rc4y^2
        Row[50]:
          Index = 49
          Value = 0.065566875
          Unit = 
          Description = m4*rc4z^2
        Row[51]:
          Index = 50
          Value = 0.037962996
          Unit = 
          Description = Jxx4
        Row[52]:
          Index = 51
          Value = 0.037962996
          Unit = 
          Description = Jyy4
        Row[53]:
          Index = 52
          Unit = 
          Description = Jzz4
        Row[54]:
          Index = 53
          Value = 0.363
          Unit = 
          Description = m5
        Row[55]:
          Index = 54
          Unit = 
          Description = m5*rc5x
        Row[56]:
          Index = 55
          Unit = 
          Description = m5*rc5y
        Row[57]:
          Index = 56
          Value = 0.154275
          Unit = 
          Description = m5*rc5z
        Row[58]:
          Index = 57
          Unit = 
          Description = m5*rc5x*rc5y
        Row[59]:
          Index = 58
          Unit = 
          Description = m5*rc5y*rc5z
        Row[60]:
          Index = 59
          Unit = 
          Description = m5*rc5x*rc5z
        Row[61]:
          Index = 60
          Unit = 
          Description = m5*rc5x^2
        Row[62]:
          Index = 61
          Unit = 
          Description = m5*rc5y^2
        Row[63]:
          Index = 62
          Value = 0.065566875
          Unit = 
          Description = m5*rc5z^2
        Row[64]:
          Index = 63
          Value = 0.037962996
          Unit = 
          Description = Jxx5
        Row[65]:
          Index = 64
          Value = 0.037962996
          Unit = 
          Description = Jyy5
        Row[66]:
          Index = 65
          Unit = 
          Description = Jzz5
        Row[67]:
          Index = 66
          Value = 0.363
          Unit = 
          Description = m6
        Row[68]:
          Index = 67
          Unit = 
          Description = m6*rc6x
        Row[69]:
          Index = 68
          Unit = 
          Description = m6*rc6y
        Row[70]:
          Index = 69
          Value = 0.154275
          Unit = 
          Description = m6*rc6z
        Row[71]:
          Index = 70
          Unit = 
          Description = m6*rc6x*rc6y
        Row[72]:
          Index = 71
          Unit = 
          Description = m6*rc6y*rc6z
        Row[73]:
          Index = 72
          Unit = 
          Description = m6*rc6x*rc6z
        Row[74]:
          Index = 73
          Unit = 
          Description = m6*rc6x^2
        Row[75]:
          Index = 74
          Unit = 
          Description = m6*rc6y^2
        Row[76]:
          Index = 75
          Value = 0.065566875
          Unit = 
          Description = m6*rc6z^2
        Row[77]:
          Index = 76
          Value = 0.037962996
          Unit = 
          Description = Jxx6
        Row[78]:
          Index = 77
          Value = 0.037962996
          Unit = 
          Description = Jyy6
        Row[79]:
          Index = 78
          Unit = 
          Description = Jzz6
        Row[80]:
          Index = 79
          Value = 0.522
          Unit = 
          Description = m7
        Row[81]:
          Index = 80
          Unit = 
          Description = m7*rc7x
        Row[82]:
          Index = 81
          Unit = 
          Description = m7*rc7y
        Row[83]:
          Index = 82
          Value = 0.13188852
          Unit = 
          Description = m7*rc7z
        Row[84]:
          Index = 83
          Unit = 
          Description = m7*rc7x*rc7y
        Row[85]:
          Index = 84
          Unit = 
          Description = m7*rc7y*rc7z
        Row[86]:
          Index = 85
          Unit = 
          Description = m7*rc7x*rc7z
        Row[87]:
          Index = 86
          Unit = 
          Description = m7*rc7x^2
        Row[88]:
          Index = 87
          Unit = 
          Description = m7*rc7y^2
        Row[89]:
          Index = 88
          Value = 0.0333229534632
          Unit = 
          Description = m7*rc7z^2
        Row[90]:
          Index = 89
          Value = 0.027879775000000002
          Unit = 
          Description = Jxx7
        Row[91]:
          Index = 90
          Value = 0.027879775000000002
          Unit = 
          Description = Jyy7
        Row[92]:
          Index = 91
          Value = 0.0019875
          Unit = 
          Description = Jzz7
        Row[93]:
          Index = 92
          Value = 0.517
          Unit = 
          Description = m8
        Row[94]:
          Index = 93
          Unit = 
          Description = m8*rc8x
        Row[95]:
          Index = 94
          Unit = 
          Description = m8*rc8y
        Row[96]:
          Index = 95
          Value = 0.12433333
          Unit = 
          Description = m8*rc8z
        Row[97]:
          Index = 96
          Unit = 
          Description = m8*rc8x*rc8y
        Row[98]:
          Index = 97
          Unit = 
          Description = m8*rc8y*rc8z
        Row[99]:
          Index = 98
          Unit = 
          Description = m8*rc8x*rc8z
        Row[100]:
          Index = 99
          Unit = 
          Description = m8*rc8x^2
        Row[101]:
          Index = 100
          Unit = 
          Description = m8*rc8y^2
        Row[102]:
          Index = 101
          Value = 0.029900922531700003
          Unit = 
          Description = m8*rc8z^2
        Row[103]:
          Index = 102
          Value = 0.026641308000000002
          Unit = 
          Description = Jxx8
        Row[104]:
          Index = 103
          Value = 0.026641308000000002
          Unit = 
          Description = Jyy8
        Row[105]:
          Index = 104
          Value = 0.0009030400000000001
          Unit = 
          Description = Jzz8
        Row[106]:
          Index = 105
          Value = 0.44
          Unit = 
          Description = m9
        Row[107]:
          Index = 106
          Unit = 
          Description = m9*rc9x
        Row[108]:
          Index = 107
          Unit = 
          Description = m9*rc9y
        Row[109]:
          Index = 108
          Unit = 
          Description = m9*rc9z
        Row[110]:
          Index = 109
          Unit = 
          Description = m9*rc9x*rc9y
        Row[111]:
          Index = 110
          Unit = 
          Description = m9*rc9y*rc9z
        Row[112]:
          Index = 111
          Unit = 
          Description = m9*rc9x*rc9z
        Row[113]:
          Index = 112
          Unit = 
          Description = m9*rc9x^2
        Row[114]:
          Index = 113
          Unit = 
          Description = m9*rc9y^2
        Row[115]:
          Index = 114
          Unit = 
          Description = m9*rc9z^2
        Row[116]:
          Index = 115
          Unit = 
          Description = Jxx9
        Row[117]:
          Index = 116
          Unit = 
          Description = Jyy9
        Row[118]:
          Index = 117
          Unit = 
          Description = Jzz9
        Row[119]:
          Index = 118
          Unit = 
          Description = m10
        Row[120]:
          Index = 119
          Unit = 
          Description = m10*rc10x
        Row[121]:
          Index = 120
          Unit = 
          Description = m10*rc10y
        Row[122]:
          Index = 121
          Unit = 
          Description = m10*rc10z
        Row[123]:
          Index = 122
          Unit = 
          Description = m10*rc10x*rc10y
        Row[124]:
          Index = 123
          Unit = 
          Description = m10*rc10y*rc10z
        Row[125]:
          Index = 124
          Unit = 
          Description = m10*rc10x*rc10z
        Row[126]:
          Index = 125
          Unit = 
          Description = m10*rc10x^2
        Row[127]:
          Index = 126
          Unit = 
          Description = m10*rc10y^2
        Row[128]:
          Index = 127
          Unit = 
          Description = m10*rc10z^2
        Row[129]:
          Index = 128
          Unit = 
          Description = Jxx10
        Row[130]:
          Index = 129
          Unit = 
          Description = Jyy10
        Row[131]:
          Index = 130
          Value = 0.00133136
          Unit = 
          Description = Jzz10
        Row[132]:
          Index = 144
          Value = 0.0003952
          Unit = 
          Description = JDrive1
        Row[133]:
          Index = 145
          Value = 0.0003952
          Unit = 
          Description = JDrive2
        Row[134]:
          Index = 146
          Value = 0.0003952
          Unit = 
          Description = JDrive3
        Row[135]:
          Index = 147
          Value = 9.24e-05
          Unit = 
          Description = JDrive4
        Row[136]:
          Index = 148
          Value = 0.24955495076809192
          Unit = 
          Description = dV1
        Row[137]:
          Index = 149
          Value = 0.24955495076809192
          Unit = 
          Description = dV2
        Row[138]:
          Index = 150
          Value = 0.24955495076809192
          Unit = 
          Description = dV3
        Row[139]:
          Index = 151
          Value = 0.060478878374920234
          Unit = 
          Description = dV4
        Row[140]:
          Index = 152
          Value = 6.16
          Unit = 
          Description = dC1
        Row[141]:
          Index = 153
          Value = 6.16
          Unit = 
          Description = dC2
        Row[142]:
          Index = 154
          Value = 6.16
          Unit = 
          Description = dC3
        Row[143]:
          Index = 155
          Value = 0.7000000000000001
          Unit = 
          Description = dC4
      InternalDynamicLimits = Used
        TypeIsReadOnly = 1
        Type = D4-ST21-1100-R11
        GearboxLimits:
          Row[1]:
            Value = 4
            Unit = Variant
            Description = Type of dynamic model
          Row[2]:
            Index = 1
            Value = 78.0
            Unit = Nm
            Description = Gearbox Drive 1 Output Torque Limit
          Row[3]:
            Index = 2
            Value = 78.0
            Unit = Nm
            Description = Gearbox Drive 2 Output Torque Limit
          Row[4]:
            Index = 3
            Value = 78.0
            Unit = Nm
            Description = Gearbox Drive 3 Output Torque Limit
          Row[5]:
            Index = 4
            Value = 4.0
            Unit = Nm
            Description = Gearbox Drive 4 Output Torque Limit
        CrossSectionLimits:
          Row[1]:
            Value = 4
            Unit = Variant
            Description = Type of dynamic model
          Row[2]:
            Index = 1
            Value = 10000.0
            Unit = N
            Description = 
          Row[3]:
            Index = 2
            Value = 10000.0
            Unit = N
            Description = 
          Row[4]:
            Index = 3
            Value = 10000.0
            Unit = N
            Description = 
          Row[5]:
            Index = 4
            Value = 10000.0
            Unit = Nm
            Description = 
          Row[6]:
            Index = 5
            Value = 10000.0
            Unit = Nm
            Description = 
          Row[7]:
            Index = 6
            Value = 10000.0
            Unit = Nm
            Description = 
          Row[8]:
            Index = 7
            Value = 150.0
            Unit = N
            Description = 
          Row[9]:
            Index = 8
            Value = 150.0
            Unit = N
            Description = 
          Row[10]:
            Index = 9
            Value = 150.0
            Unit = N
            Description = 
          Row[11]:
            Index = 10
            Value = 150.0
            Unit = N
            Description = 
          Row[12]:
            Index = 11
            Value = 150.0
            Unit = N
            Description = 
          Row[13]:
            Index = 12
            Value = 150.0
            Unit = N
            Description = 
      LoadDependentJerkLimitsIsReadOnly = 1
      LoadDependentJerkLimits = PayloadDependentJerkReduction
        JerkReduction[1]:
          PayloadInKgIsReadOnly = 1
          PayloadInKg = 0.0
          JerkReductionInPercentIsReadOnly = 1
          JerkReductionInPercent = 0.0
        JerkReduction[2]:
          PayloadInKgIsReadOnly = 1
          PayloadInKg = 0.35
          JerkReductionInPercentIsReadOnly = 1
          JerkReductionInPercent = 0.0
        JerkReduction[3]:
          PayloadInKgIsReadOnly = 1
          PayloadInKg = 1.0
          JerkReductionInPercentIsReadOnly = 1
          JerkReductionInPercent = 50.0
        JerkReduction[4]:
          PayloadInKgIsReadOnly = 1
          PayloadInKg = 2.0
          JerkReductionInPercentIsReadOnly = 1
          JerkReductionInPercent = 50.0
        JerkReduction[5]:
          PayloadInKgIsReadOnly = 1
          PayloadInKg = 3.0
          JerkReductionInPercentIsReadOnly = 1
          JerkReductionInPercent = 75.0
      JointAxesPositionLimits:
        JointAxisIsReadOnly = 1
        JointAxis[1]
        JointAxis[2]
        JointAxis[3]
        JointAxis[4]
      WorkingRangeIsReadOnly = 1
      WorkingRange = Standard
        BaseToTopIsReadOnly = 1
        BaseToTop = 710.0
        TopHeightIsReadOnly = 1
        MiddleHeightIsReadOnly = 1
        MiddleHeight = 250.0
        BottomHeightIsReadOnly = 1
        BottomHeight = 210.0
        TopRadiusIsReadOnly = 1
        TopRadius = 550.0
        MiddleRadiusIsReadOnly = 1
        MiddleRadius = 550.0
        BottomRadiusIsReadOnly = 1
        BottomRadius = 150.0
```

### Config_11.axesgroupfeature - 5APC3100_KBU3_000/mappMotion/Robots/Codian_D4r1100R_2/Config_11.axesgroupfeature
```
Element Feature_Programs_D4r1100R_2 (Type=axesgroupfeature)
  Type:
    ProgramElements:
      PVs:
        PV[1]:
          PvName = ::MovePrg:GripperRobot2OpenClose
          Advanced:
            Alias = CloseGripper
            Synchronization = Path
```

### Config_8.axesgroup - 5APC3100_KBU3_000/mappMotion/Robots/Codian_D4r1100R_2/Config_8.axesgroup
```
Element gAxesGroup_D4r1100R_2 (Type=axesgroup)
  Type = PathGenAxesGroup
    ProcessingTaskClass = 1
    PhysicalAxes:
      JointAxes:
        JointAxis[1]:
          AxisRef = gAxisQ1_D4r1100R_2
        JointAxis[2]:
          AxisRef = gAxisQ2_D4r1100R_2
        JointAxis[3]:
          AxisRef = gAxisQ3_D4r1100R_2
        JointAxis[4]:
          Name = QC
          AxisRef = gAxisQC_D4r1100R_2
    MechanicalSystem:
      MechSysRef = MechSys_D4r1100R_2
    BasicSettings:
      GeometryPlanning:
        MaxTangentialTransitionDeviation = 0.05
      TrajectoryPlanning:
        LimitCheckResolution:
          Time = 0.005
        BufferTime:
          Time = 0.05
      Miscellaneous:
        TimeStretchOverride:
          JerkSuppression = Basic
            AdaptationTime = 0.3
    StopReaction:
      AxisError:
        AxisReaction = DynamicStop
    AxesGroupFeatures:
      FeatureRef[1] = Feature_Programs_D4r1100R_2
      FeatureRef[2] = Feature_FeedForward_D4r1100R_X
      FeatureRef[3] = Feature_Jogging_D4r1100R_X
      FeatureRef[4] = Feature_PathDefinitions_D4r1100R_X
      FeatureRef[5] = Feature_Tracking_D4r1100R_X
      FeatureRef[6] = Feature_TrkFrmSel_D4r1100R_X
```

### Config_9.axis - 5APC3100_KBU3_000/mappMotion/Robots/Codian_D4r1100R_2/Config_9.axis
```
Element gAxisQ1_D4r1100R_2 (Type=axis)
  BaseTypeIsReadOnly = 1
  BaseType = RotaryBounded
    MeasurementUnitIsReadOnly = 1
    MeasurementResolutionIsReadOnly = 1
    MeasurementResolution = 0.001
    CountDirectionIsReadOnly = 1
    CountDirection = Inverse
  MovementLimits = InternalForPathControlledAxis
    Position:
      LowerLimitMin = -46.0
      UpperLimitMax = 101.0
      LowerLimit = -46.0
      UpperLimit = 101.0
    Velocity:
      VelocityMax = 680.0
      Velocity = 680.0
    Acceleration:
      AccelerationMax = 35000.0
      Acceleration = 35000.0
    Deceleration:
      DecelerationMax = 35000.0
      Deceleration = 35000.0
    Jerk = Advanced
      JerkAccelerationPositiveMin = 0.0
      JerkAccelerationPositiveMax = 4200000.0
      JerkAccelerationPositive = 4200000.0
      JerkAccelerationNegativeMin = 0.0
      JerkAccelerationNegativeMax = 4200000.0
      JerkAccelerationNegative = 4200000.0
      JerkDecelerationPositiveMin = 0.0
      JerkDecelerationPositiveMax = 3200000.0
      JerkDecelerationPositive = 3200000.0
      JerkDecelerationNegativeMin = 0.0
      JerkDecelerationNegativeMax = 3200000.0
      JerkDecelerationNegative = 3200000.0
    Torque = Basic
      TorqueMax = 11.0
      Torque = 11.0
Element gAxisQ2_D4r1100R_2 (Type=axis)
  BaseTypeIsReadOnly = 1
  BaseType = RotaryBounded
    MeasurementUnitIsReadOnly = 1
    MeasurementResolutionIsReadOnly = 1
    MeasurementResolution = 0.001
    CountDirectionIsReadOnly = 1
    CountDirection = Inverse
  MovementLimits = InternalForPathControlledAxis
    Position:
      LowerLimitMin = -46.0
      UpperLimitMax = 101.0
      LowerLimit = -46.0
      UpperLimit = 101.0
    Velocity:
      VelocityMax = 680.0
      Velocity = 680.0
    Acceleration:
      AccelerationMax = 35000.0
      Acceleration = 35000.0
    Deceleration:
      DecelerationMax = 35000.0
      Deceleration = 35000.0
    Jerk = Advanced
      JerkAccelerationPositiveMin = 0.0
      JerkAccelerationPositiveMax = 4200000.0
      JerkAccelerationPositive = 4200000.0
      JerkAccelerationNegativeMin = 0.0
      JerkAccelerationNegativeMax = 4200000.0
      JerkAccelerationNegative = 4200000.0
      JerkDecelerationPositiveMin = 0.0
      JerkDecelerationPositiveMax = 3200000.0
      JerkDecelerationPositive = 3200000.0
      JerkDecelerationNegativeMin = 0.0
      JerkDecelerationNegativeMax = 3200000.0
      JerkDecelerationNegative = 3200000.0
    Torque = Basic
      TorqueMax = 11.0
      Torque = 11.0
Element gAxisQ3_D4r1100R_2 (Type=axis)
  BaseTypeIsReadOnly = 1
  BaseType = RotaryBounded
    MeasurementUnitIsReadOnly = 1
    MeasurementResolutionIsReadOnly = 1
    MeasurementResolution = 0.001
    CountDirectionIsReadOnly = 1
    CountDirection = Inverse
  MovementLimits = InternalForPathControlledAxis
    Position:
      LowerLimitMin = -46.0
      UpperLimitMax = 101.0
      LowerLimit = -46.0
      UpperLimit = 101.0
    Velocity:
      VelocityMax = 680.0
      Velocity = 680.0
    Acceleration:
      AccelerationMax = 35000.0
      Acceleration = 35000.0
    Deceleration:
      DecelerationMax = 35000.0
      Deceleration = 35000.0
    Jerk = Advanced
      JerkAccelerationPositiveMin = 0.0
      JerkAccelerationPositiveMax = 4200000.0
      JerkAccelerationPositive = 4200000.0
      JerkAccelerationNegativeMin = 0.0
      JerkAccelerationNegativeMax = 4200000.0
      JerkAccelerationNegative = 4200000.0
      JerkDecelerationPositiveMin = 0.0
      JerkDecelerationPositiveMax = 3200000.0
      JerkDecelerationPositive = 3200000.0
      JerkDecelerationNegativeMin = 0.0
      JerkDecelerationNegativeMax = 3200000.0
      JerkDecelerationNegative = 3200000.0
    Torque = Basic
      TorqueMax = 11.0
      Torque = 11.0
Element gAxisQC_D4r1100R_2 (Type=axis)
  BaseTypeIsReadOnly = 1
  BaseType = Rotary
    MeasurementUnitIsReadOnly = 1
    MeasurementResolutionIsReadOnly = 1
    MeasurementResolution = 0.001
    CountDirectionIsReadOnly = 1
  MovementLimits = InternalForPathControlledAxis
    Velocity:
      VelocityMax = 3600.0
      Velocity = 3600.0
    Acceleration:
      AccelerationMax = 75000.0
      Acceleration = 75000.0
    Deceleration:
      DecelerationMax = 75000.0
      Deceleration = 75000.0
    Jerk = Advanced
      JerkAccelerationPositiveMin = 0.0
      JerkAccelerationPositiveMax = 10000000.0
      JerkAccelerationPositive = 10000000.0
      JerkAccelerationNegativeMin = 0.0
      JerkAccelerationNegativeMax = 10000000.0
      JerkAccelerationNegative = 10000000.0
      JerkDecelerationPositiveMin = 0.0
      JerkDecelerationPositiveMax = 10000000.0
      JerkDecelerationPositive = 10000000.0
      JerkDecelerationNegativeMin = 0.0
      JerkDecelerationNegativeMax = 10000000.0
      JerkDecelerationNegative = 10000000.0
    Torque = Basic
      TorqueMax = 4.0
      Torque = 4.0
```

### CommonFeat.axesgroupfeature - 5APC3100_KBU3_000/mappMotion/Robots/CommonFeat.axesgroupfeature
```
Element Feature_FeedForward_D4r1100R_X (Type=axesgroupfeature)
  Type = FeedForward
    RiseTime = 0.25
    Filter = AxisJerkTime
Element Feature_Jogging_D4r1100R_X (Type=axesgroupfeature)
  Type = Jogging
Element Feature_Tracking_D4r1100R_X (Type=axesgroupfeature)
  Type = Tracking
    MotionBehaviour:
      OutOfWorkspaceSynchronisation:
        Clearance = 50
Element Feature_PathDefinitions_D4r1100R_X (Type=axesgroupfeature)
  Type = PathDefinitions
    PathDefinition[1]:
      Type:
        CalculatedIn = PCS
Element Feature_TrkFrmSel_D4r1100R_X (Type=axesgroupfeature)
  Type = TrackingFrameSelection
    Selectors:
      Selector[1]:
        Name = PickPositionSelector
        Filters:
          Filter[1]:
            TrackingPathRef[1] = gTrkPath_Conveyor_1
          Filter[2] = SelectionArea
            Area[1] = Cylinder
              Translation:
                X = -500
                Z = -992.6
              Dimensions:
                Radius = 500
                Height = 250
        LockingAfterSelection = AllSelectors
      Selector[2]:
        Name = PlacePositionSelector
        Filters:
          Filter[1]:
            TrackingPathRef[1] = gTrkPath_Conveyor_2
          Filter[2] = SelectionArea
            Area[1] = Cylinder
              Translation:
                X = -500
                Z = -992.6
              Dimensions:
                Radius = 500
                Height = 250
        LockingAfterSelection = AllSelectors
```

## Logical view

Binary libraries used (declarations not repeated): operator, runtime, AsIecCon, astime, MpBase, McBase, MpAxis, McAcpAx, McPathGen, McPureVAx, McAxGroup, McAxis, McProgInt, McTrkPath, MpRobotics


### Program Logical/MovePrg (IEC) - Power, Home, Move 

#### Types.typ
```iecst
TYPE
	CommandType : 	STRUCT
		PowerAndHome : BOOL;
		MoveConveyor1 : BOOL;
		MoveConveyor2 : BOOL;
		MoveProgramRobot1 : BOOL;
		MoveProgramRobot2 : BOOL;
		Settings : CmdSettingsType;
	END_STRUCT;
	CmdSettingsType : 	STRUCT
		FrameSpaceConveyor1 : LREAL;
		FrameSpaceConveyor2 : LREAL;
		VelocityConveyor1 : REAL;
		VelocityConveyor2 : REAL;
	END_STRUCT;
	StateType :
		(
		STARTUP,
		WAIT_FOR_POWER_AND_HOME,
		POWER,
		HOME,
		READ_CURRENT_PARAMETERS,
		RUN
		);
END_TYPE
```

#### Variables.var
```iecst
(*Command interface*)
VAR
	Cmd : CommandType;
END_VAR
(*Robot and conveyor FBs*)
VAR
	MpRobot_0 : MpDelta4Axis;
	MpRobot_1 : MpDelta4Axis;
	MpRobotPar : MpDelta4AxisParType;
	MpAxisConv1 : MpAxisBasic;
	MpAxisConv2 : MpAxisBasic;
	MpAxisParConv1 : MpAxisBasicParType;
	MpAxisParConv2 : MpAxisBasicParType;
END_VAR
(*Update automatic TrackingFrame creation*)
VAR
	ProcessParam_AutCrtCond1TrkPath1 : MC_BR_ProcessParam;
	ProcessParam_AutCrtCond1TrkPath2 : MC_BR_ProcessParam;
	AutoCreateConditionParTrkPath1 : McCfgTrkPathAutCrtCondType;
	AutoCreateConditionParTrkPath2 : McCfgTrkPathAutCrtCondType;
	StatusTrackingPath1 : MC_BR_TrackingPathReadStatus;
	StatusTrackingPath2 : MC_BR_TrackingPathReadStatus;
END_VAR
(*State machine*)
VAR
	State : StateType;
END_VAR
(*Grippers*)
VAR
	GripperRobot1OpenClose : BOOL;
	GripperRobot2OpenClose : BOOL;
END_VAR
(*Optional manual TrackingFrame creation*)
VAR
	MC_BR_TrackingFrameCreate_0 : MC_BR_TrackingFrameCreate;
	ManualCreationTrigger : BOOL;
END_VAR
```

#### Main.st
```iecst
PROGRAM _INIT

	//Initial process parameters
	Cmd.Settings.FrameSpaceConveyor1 := 150;
	Cmd.Settings.FrameSpaceConveyor2 := 150;
	Cmd.Settings.VelocityConveyor1 := 400;
	Cmd.Settings.VelocityConveyor2 := 400;

	// Robots
	MpRobotPar.ProgramName := 'pnpPrg.st';
	MpRobot_0.MpLink := ADR(gAxesGroup_D4r1100R_1);
	MpRobot_0.Enable := TRUE;
	MpRobot_0.Parameters := ADR(MpRobotPar);
	MpRobot_0.Override := 100;
	MpRobot_1.MpLink := ADR(gAxesGroup_D4r1100R_2);
	MpRobot_1.Enable := TRUE;
	MpRobot_1.Parameters := ADR(MpRobotPar);
	MpRobot_1.Override := 100;

	// Conveyor belts
	MpAxisParConv1.Velocity := Cmd.Settings.VelocityConveyor1;
	MpAxisParConv2.Velocity := Cmd.Settings.VelocityConveyor2;
	MpAxisConv1.MpLink := ADR(gAxis_Conveyor_1);
	MpAxisConv1.Parameters := ADR(MpAxisParConv1);
	MpAxisConv1.Enable := TRUE;
	MpAxisConv2.MpLink := ADR(gAxis_Conveyor_2);
	MpAxisConv2.Parameters := ADR(MpAxisParConv2);
	MpAxisConv2.Enable := TRUE;
	StatusTrackingPath1.Enable := TRUE;
	StatusTrackingPath2.Enable := TRUE;
	StatusTrackingPath1.TrackingPath := ADR(gTrkPath_Conveyor_1);
	StatusTrackingPath2.TrackingPath := ADR(gTrkPath_Conveyor_2);

	GripperRobot1OpenClose := FALSE; // Open
	GripperRobot2OpenClose := FALSE; // Open

	gAxisQ1_D4r1100R_1;
	gAxisQ2_D4r1100R_1;
	gAxisQ3_D4r1100R_1;
	gAxisQC_D4r1100R_1;

	gAxisQ1_D4r1100R_2;
	gAxisQ2_D4r1100R_2;
	gAxisQ3_D4r1100R_2;
	gAxisQC_D4r1100R_2;

END_PROGRAM

PROGRAM _CYCLIC

	// User Interface update
	MpRobot_0.MoveProgram := Cmd.MoveProgramRobot1;
	MpRobot_1.MoveProgram := Cmd.MoveProgramRobot2;
	MpAxisConv1.MoveVelocity := Cmd.MoveConveyor1;
	MpAxisConv2.MoveVelocity := Cmd.MoveConveyor2;

	// Main state machine
	CASE State OF

		STARTUP:

			IF MpRobot_0.Info.ReadyToPowerOn AND MpRobot_1.Info.ReadyToPowerOn AND MpAxisConv1.Info.ReadyToPowerOn AND MpAxisConv2.Info.ReadyToPowerOn THEN
				State := WAIT_FOR_POWER_AND_HOME;
			END_IF

		WAIT_FOR_POWER_AND_HOME:

			// AxesGroups are still disabled in this state and optionally ProcessParam_TrkFrmSelectionFeat FB can be used to manually manipulate the configured parameters
			IF Cmd.PowerAndHome THEN
				State := POWER;
			END_IF

		POWER:

			MpRobot_0.Power := TRUE;
			MpRobot_1.Power := TRUE;
			MpAxisConv1.Power := TRUE;
			MpAxisConv2.Power := TRUE;
			IF MpRobot_0.PowerOn AND MpRobot_1.PowerOn  AND MpAxisConv1.PowerOn AND MpAxisConv2.PowerOn THEN
				State := HOME;
			END_IF

		HOME:

			MpRobot_0.Home := TRUE;
			MpRobot_1.Home := TRUE;
			MpAxisConv1.Home := TRUE;
			MpAxisConv2.Home := TRUE;
			IF MpRobot_0.IsHomed AND MpRobot_1.IsHomed AND MpAxisConv1.IsHomed AND MpAxisConv2.IsHomed THEN
				State := READ_CURRENT_PARAMETERS;
			END_IF

		READ_CURRENT_PARAMETERS:

			// Read current automatic creation condition parameters configured for TrackingPath components

			IF StatusTrackingPath1.TrackingPathReady AND StatusTrackingPath2.TrackingPathReady THEN
				ProcessParam_AutCrtCond1TrkPath1.Execute := TRUE;
				ProcessParam_AutCrtCond1TrkPath1.Component := ADR(gTrkPath_Conveyor_1);
				ProcessParam_AutCrtCond1TrkPath1.AdvancedParameters.Name := 'Condition 1';
				ProcessParam_AutCrtCond1TrkPath1.DataAddress := ADR(AutoCreateConditionParTrkPath1);
				ProcessParam_AutCrtCond1TrkPath1.DataType := mcCFG_TRK_PATH_AUT_CRT_COND;
				ProcessParam_AutCrtCond1TrkPath1.Mode := mcPPM_READ;

				ProcessParam_AutCrtCond1TrkPath2.Execute := TRUE;
				ProcessParam_AutCrtCond1TrkPath2.Component := ADR(gTrkPath_Conveyor_2);
				ProcessParam_AutCrtCond1TrkPath2.AdvancedParameters.Name := 'Condition 1';
				ProcessParam_AutCrtCond1TrkPath2.DataAddress := ADR(AutoCreateConditionParTrkPath2);
				ProcessParam_AutCrtCond1TrkPath2.DataType := mcCFG_TRK_PATH_AUT_CRT_COND;
				ProcessParam_AutCrtCond1TrkPath2.Mode := mcPPM_READ;
			END_IF

			IF ProcessParam_AutCrtCond1TrkPath1.Done AND ProcessParam_AutCrtCond1TrkPath2.Done THEN

				ProcessParam_AutCrtCond1TrkPath1.Execute := FALSE;
				ProcessParam_AutCrtCond1TrkPath2.Execute := FALSE;

				Cmd.Settings.FrameSpaceConveyor1 := AutoCreateConditionParTrkPath1.Condition.DistanceBased.Distance;
				Cmd.Settings.FrameSpaceConveyor2 := AutoCreateConditionParTrkPath2.Condition.DistanceBased.Distance;

				State := RUN;

			END_IF

		RUN:

			// Update with commanded automatic TrackingFrame creation parameters
			IF AutoCreateConditionParTrkPath1.Condition.DistanceBased.Distance <> Cmd.Settings.FrameSpaceConveyor1 THEN
				AutoCreateConditionParTrkPath1.Condition.DistanceBased.Distance := Cmd.Settings.FrameSpaceConveyor1;
				ProcessParam_AutCrtCond1TrkPath1.Execute := TRUE;
				ProcessParam_AutCrtCond1TrkPath1.Component := ADR(gTrkPath_Conveyor_1);
				ProcessParam_AutCrtCond1TrkPath1.AdvancedParameters.Name := 'Condition 1';
				ProcessParam_AutCrtCond1TrkPath1.DataAddress := ADR(AutoCreateConditionParTrkPath1);
				ProcessParam_AutCrtCond1TrkPath1.DataType := mcCFG_TRK_PATH_AUT_CRT_COND;
				ProcessParam_AutCrtCond1TrkPath1.Mode := mcPPM_WRITE;
				ProcessParam_AutCrtCond1TrkPath1();
				ProcessParam_AutCrtCond1TrkPath1.Execute := FALSE;
			END_IF
			IF AutoCreateConditionParTrkPath2.Condition.DistanceBased.Distance <> Cmd.Settings.FrameSpaceConveyor2 THEN
				AutoCreateConditionParTrkPath2.Condition.DistanceBased.Distance := Cmd.Settings.FrameSpaceConveyor2;
				ProcessParam_AutCrtCond1TrkPath2.Execute := TRUE;
				ProcessParam_AutCrtCond1TrkPath2.Component := ADR(gTrkPath_Conveyor_2);
				ProcessParam_AutCrtCond1TrkPath2.AdvancedParameters.Name := 'Condition 1';
				ProcessParam_AutCrtCond1TrkPath2.DataAddress := ADR(AutoCreateConditionParTrkPath2);
				ProcessParam_AutCrtCond1TrkPath2.DataType := mcCFG_TRK_PATH_AUT_CRT_COND;
				ProcessParam_AutCrtCond1TrkPath2.Mode := mcPPM_WRITE;
				ProcessParam_AutCrtCond1TrkPath2();
				ProcessParam_AutCrtCond1TrkPath2.Execute := FALSE;
			END_IF

			// Update commanded conveyor belt velocities
			IF MpAxisParConv1.Velocity <> Cmd.Settings.VelocityConveyor1 THEN
				MpAxisParConv1.Velocity := Cmd.Settings.VelocityConveyor1;
				MpAxisConv1.Update := TRUE;
				MpAxisConv1();
				MpAxisConv1.Update := FALSE;
			END_IF
			IF MpAxisParConv2.Velocity <> Cmd.Settings.VelocityConveyor2 THEN
				MpAxisParConv2.Velocity := Cmd.Settings.VelocityConveyor2;
				MpAxisConv2.Update := TRUE;
				MpAxisConv2();
				MpAxisConv2.Update := FALSE;
			END_IF

			// Optional: Application dependent creation of TrackingFrames (example)
			MC_BR_TrackingFrameCreate_0.Execute := ManualCreationTrigger;
			MC_BR_TrackingFrameCreate_0.TrackingPath := ADR(gTrkPath_Conveyor_1);
			// Position (relative to TrackingPath) at time of object detection
			MC_BR_TrackingFrameCreate_0.Parameters.Translation.X := 0;
			MC_BR_TrackingFrameCreate_0.Parameters.Translation.Y := -50;
			MC_BR_TrackingFrameCreate_0.Parameters.Translation.Z := 0;
			// Conveyor position at time of object detection
			MC_BR_TrackingFrameCreate_0.Parameters.LatchedPath.Position := MpAxisConv1.Position;
			// Wait for MC_BR_TrackingFrameCreate_0.Done
			IF (MC_BR_TrackingFrameCreate_0.Done) THEN
				ManualCreationTrigger := FALSE;
			END_IF

	END_CASE

	// Call function blocks
	MC_BR_TrackingFrameCreate_0();
	MpRobot_0();
	MpRobot_1();
	MpAxisConv1();
	MpAxisConv2();
	ProcessParam_AutCrtCond1TrkPath1();
	ProcessParam_AutCrtCond1TrkPath2();
	StatusTrackingPath1();
	StatusTrackingPath2();

END_PROGRAM
```

### Program Logical/ParChange (IEC) - Optional: Parameter changes at runtime 

#### Variables.var
```iecst
(*Change TrackingFrameSelection feature configuration/parameters*)
VAR
	ProcessParam_TrkFrmSelectionFeat : MC_BR_ProcessParam;
	TrkFrmSelConfig : McCfgAxGrpFeatTrkFrmSelType;
	TrkFrmSelConfig_Selectors : ARRAY[0..9] OF McAGFTFSSelSelType;
END_VAR
(*Selector 1*)
VAR
	TrkFrmSelConfig_Sel1Filters : ARRAY[0..1] OF McAGFTFSSFFltrFltrType;
	TrkFrmSelConfig_Sel1Areas : ARRAY[0..1] OF McAGFTFSSFSFSAAreaType;
	TrkFrmSelConfig_Sel1TrkPaths : ARRAY[0..1] OF McCfgReferenceType;
END_VAR
(*Selector 2*)
VAR
	TrkFrmSelConfig_Sel2Filters : ARRAY[0..1] OF McAGFTFSSFFltrFltrType;
	TrkFrmSelConfig_Sel2Areas : ARRAY[0..1] OF McAGFTFSSFSFSAAreaType;
	TrkFrmSelConfig_Sel2TrkPaths : ARRAY[0..1] OF McCfgReferenceType;
END_VAR
```

#### Main.st
```iecst
PROGRAM _INIT

	// ------------------------------------------------------------------------------------------------
	// Optional: Operate on parameters of TrackingFrameSelection feature for robot 1 during PLC runtime

	// ------------------------------------------------------------------------------------------------
	// Prepare dummy parameters and data type with 'unbounded arrays'

	// AxesGroupFeature - TrackingFrameSelection - Parmeters
	// Selectors
	TrkFrmSelConfig.Selectors.Selector.DataAddress := ADR(TrkFrmSelConfig_Selectors);
	TrkFrmSelConfig.Selectors.Selector.NumberOfArrayElements := 10;
	TrkFrmSelConfig.Selectors.Selector.NumberOfElements := 2;
	// Selector 1
	TrkFrmSelConfig_Selectors[0].Type := mcAGFTFSSS_SNG_FRM;
	TrkFrmSelConfig_Selectors[0].SingleFrames.Name := 'myTrkFrmSelector2';
	// Selector 1 - Strategy
	TrkFrmSelConfig_Selectors[0].SingleFrames.Strategy.Type := mcAGFTFSSFS_FIFO;
	// Selector 1 - Filters
	TrkFrmSelConfig_Selectors[0].SingleFrames.Filters.Filter.DataAddress := ADR(TrkFrmSelConfig_Sel1Filters);
	TrkFrmSelConfig_Selectors[0].SingleFrames.Filters.Filter.NumberOfArrayElements := 2;
	TrkFrmSelConfig_Selectors[0].SingleFrames.Filters.Filter.NumberOfElements := 2;
	// Selector 1 - First filter - Specific tracking path
	TrkFrmSelConfig_Sel1Filters[0].TrackingPaths.TrackingPathReference.DataAddress := ADR(TrkFrmSelConfig_Sel1TrkPaths);
	TrkFrmSelConfig_Sel1Filters[0].TrackingPaths.TrackingPathReference.NumberOfArrayElements := 2;
	TrkFrmSelConfig_Sel1Filters[0].TrackingPaths.TrackingPathReference.NumberOfElements := 2;
	// Selector 1 - Second filter - Selection area
	TrkFrmSelConfig_Sel1Filters[1].SelectionArea.Area.DataAddress := ADR(TrkFrmSelConfig_Sel1Areas);
	TrkFrmSelConfig_Sel1Filters[1].SelectionArea.Area.NumberOfArrayElements := 2;
	TrkFrmSelConfig_Sel1Filters[1].SelectionArea.Area.NumberOfElements := 1;
	// Selector 1 - TrackingPaths
	TrkFrmSelConfig_Sel1TrkPaths[0].ConfigType := mcCFG_TRK_PATH;
	TrkFrmSelConfig_Sel1TrkPaths[0].Name := 'gTrkPath_Conveyor_1';
	// Selector 1 - Selection area
	TrkFrmSelConfig_Sel1Areas[0].Type := mcAGFTFSSFSFSAA_CYLINDER;
	TrkFrmSelConfig_Sel1Areas[0].Cylinder.Dimensions.Radius := 500;
	TrkFrmSelConfig_Sel1Areas[0].Cylinder.Dimensions.Height := 300;
	TrkFrmSelConfig_Sel1Areas[0].Cylinder.Origin.Type := mcAGFTFSSFSFSAACylO_MCS;
	TrkFrmSelConfig_Sel1Areas[0].Cylinder.Orientation.Angle1:= 0;
	TrkFrmSelConfig_Sel1Areas[0].Cylinder.Orientation.Angle2:= 0;
	TrkFrmSelConfig_Sel1Areas[0].Cylinder.Orientation.Angle3:= 0;
	TrkFrmSelConfig_Sel1Areas[0].Cylinder.Translation.X := -300;
	TrkFrmSelConfig_Sel1Areas[0].Cylinder.Translation.Y := 0;
	TrkFrmSelConfig_Sel1Areas[0].Cylinder.Translation.Z := -100;
	// Selector 2
	TrkFrmSelConfig_Selectors[1].Type := mcAGFTFSSS_SNG_FRM;
	TrkFrmSelConfig_Selectors[1].SingleFrames.Name := 'myTrkFrmSelector1';
	// Selector 2 - Strategy
	TrkFrmSelConfig_Selectors[1].SingleFrames.Strategy.Type := mcAGFTFSSFS_FIFO;
	// Selector 2 - Filters
	TrkFrmSelConfig_Selectors[1].SingleFrames.Filters.Filter.DataAddress := ADR(TrkFrmSelConfig_Sel2Filters);
	TrkFrmSelConfig_Selectors[1].SingleFrames.Filters.Filter.NumberOfArrayElements := 2;
	TrkFrmSelConfig_Selectors[1].SingleFrames.Filters.Filter.NumberOfElements := 2;
	// Selector 2 - First filter - Specific tracking path
	TrkFrmSelConfig_Sel2Filters[0].TrackingPaths.TrackingPathReference.DataAddress := ADR(TrkFrmSelConfig_Sel2TrkPaths);
	TrkFrmSelConfig_Sel2Filters[0].TrackingPaths.TrackingPathReference.NumberOfArrayElements := 2;
	TrkFrmSelConfig_Sel2Filters[0].TrackingPaths.TrackingPathReference.NumberOfElements := 2;
	// Selector 2 - Second filter - Selection area
	TrkFrmSelConfig_Sel2Filters[1].SelectionArea.Area.DataAddress := ADR(TrkFrmSelConfig_Sel2Areas);
	TrkFrmSelConfig_Sel2Filters[1].SelectionArea.Area.NumberOfArrayElements := 2;
	TrkFrmSelConfig_Sel2Filters[1].SelectionArea.Area.NumberOfElements := 1;
	// Selector 2 - TrackingPaths
	TrkFrmSelConfig_Sel2TrkPaths[0].ConfigType := mcCFG_TRK_PATH;
	TrkFrmSelConfig_Sel2TrkPaths[0].Name := 'gTrkPath_Conveyor_1';
	// Selector 2 - Selection area
	TrkFrmSelConfig_Sel2Areas[0].Type := mcAGFTFSSFSFSAA_CYLINDER;
	TrkFrmSelConfig_Sel2Areas[0].Cylinder.Dimensions.Radius := 500;
	TrkFrmSelConfig_Sel2Areas[0].Cylinder.Dimensions.Height := 300;
	TrkFrmSelConfig_Sel2Areas[0].Cylinder.Origin.Type := mcAGFTFSSFSFSAACylO_MCS;
	TrkFrmSelConfig_Sel2Areas[0].Cylinder.Orientation.Angle1:= 0;
	TrkFrmSelConfig_Sel2Areas[0].Cylinder.Orientation.Angle2:= 0;
	TrkFrmSelConfig_Sel2Areas[0].Cylinder.Orientation.Angle3:= 0;
	TrkFrmSelConfig_Sel2Areas[0].Cylinder.Translation.X := -300;
	TrkFrmSelConfig_Sel2Areas[0].Cylinder.Translation.Y := 0;
	TrkFrmSelConfig_Sel2Areas[0].Cylinder.Translation.Z := -100;

	// ------------------------------------------------------------------------------------------------

	// Prepare function block for optional manual execution in Watch window
	// ...to manipulate TrackingFrameSelection parameters for robot 1
	ProcessParam_TrkFrmSelectionFeat.Component := ADR(gAxesGroup_D4r1100R_1);
	ProcessParam_TrkFrmSelectionFeat.AdvancedParameters.Name := 'Feature_TrkFrmSel_D4r1100R_X';
	ProcessParam_TrkFrmSelectionFeat.DataAddress := ADR(TrkFrmSelConfig);
	ProcessParam_TrkFrmSelectionFeat.DataType := mcCFG_AXGRP_FEAT_TRKFRM_SEL;
	ProcessParam_TrkFrmSelectionFeat.Mode := mcPPM_READ;

	// ------------------------------------------------------------------------------------------------

END_PROGRAM

PROGRAM _CYCLIC

	ProcessParam_TrkFrmSelectionFeat();

END_PROGRAM
```

### pnpPrg.st - Robot program (MotionST)
```iecst
TYPE
  MachineState : (Start, SelectPickPosition, PickObject, SelectPlacePosition, PlaceObject, ParkWithNoObject, ParkWithGrippedObject);
END_TYPE

VAR CONSTANT
    ParkPos      : McPointType := (Pos:=(X:=0, Y:=0, Z:= -900));
    SynchPosUp   : McPointType := (Pos:=(X:=   0, Y:= 0,  Z:= 100));
    SynchPosDown : McPointType := (Pos:=(X:=   0, Y:= 0,  Z:= 0));
END_VAR

VAR
    TrkFrmID_PickPosition: McTrkFrmIdentType;
    TrkFrmID_PlacePosition: McTrkFrmIdentType;
    State : MachineState;
END_VAR

PROGRAM _MAIN

    State := MachineState#Start;

    REPEAT
        CASE State OF

        MachineState#Start:
            MoveLR(ParkPos);
            WaitUntilSync(TrackingFrameIsAvailable('PickPositionSelector'));
            State := MachineState#SelectPickPosition;

        MachineState#SelectPickPosition:
            WaitALAP();
            IF TrackingFrameSelect(TrkFrmID_PickPosition, 'PickPositionSelector') THEN
                State :=  MachineState#PickObject;
            ELSE
                State := MachineState#ParkWithNoObject;
            END_IF

        MachineState#PickObject:
            TrackObjectR(TrkFrmID_PickPosition, SynchPosUp, 50, 50);
            MoveLR(SynchPosDown);
			CloseGripper := TRUE;	//close gripper
			WaitTime(0.01);			//wait until gripper is closed [s]
            MoveLR(SynchPosUp);
            State := MachineState#SelectPlacePosition;

        MachineState#SelectPlacePosition:
            WaitALAP();
            IF TrackingFrameSelect(TrkFrmID_PlacePosition, 'PlacePositionSelector') THEN
                State :=  MachineState#PlaceObject;
            ELSE
                State := MachineState#ParkWithGrippedObject;
            END_IF

        MachineState#PlaceObject:
            TrackObjectR(TrkFrmID_PlacePosition, SynchPosUp, 50, 50);
            MoveLR(SynchPosDown);
			CloseGripper := FALSE;	//open gripper
			WaitTime(0.01);			//wait until gripper is opened [s]
            MoveLR(SynchPosUp);
            State := MachineState#SelectPickPosition;

        MachineState#ParkWithNoObject:
            TrackStopR(MachineFrame, ParkPos, 50, 50);
			WaitUntilSync(TrackingFrameSelect(TrkFrmID_PickPosition, 'PickPositionSelector'));
            State := MachineState#PickObject;

        MachineState#ParkWithGrippedObject:
            TrackStopR(MachineFrame, ParkPos, 50, 50);
			WaitUntilSync(TrackingFrameSelect(TrkFrmID_PlacePosition, 'PlacePositionSelector'));
			State := MachineState#PlaceObject;

        END_CASE
    UNTIL FALSE END_REPEAT;

END_PROGRAM
```

Listed in the project but not available here: Logical/Global.typ, Logical/Global.var
